//	(* Append sample digital inputs *)
//	FOR iLoop := 0 TO 19 DO
//		fbVisuControl.MR_AppendSafeInput(ifSafeInput := stShell.stPlatform.ref_fbMachineControler.SafeInputs[iLoop]);
//	END_FOR
	
//	(* Append sample digital outputs *)
//	FOR iLoop := 0 TO 19 DO
//		fbVisuControl.MR_AppendSafeOutput(ifSafeOutput := stShell.stPlatform.ref_fbMachineControler.SafeOutputs[iLoop]);
//	END_FOR
	
//	(* Append sample double coil cylinders *)
//	FOR iLoop := 0 TO 9 DO
//		fbVisuControl.MR_AppendCylinder( 	ifCylinder 			:= stShell.stPlatform.ref_fbMachineControler.DoubleCoilCylinders[iLoop],
//											eCylinderType 		:= CYLINDER_TYPE_DOUBLE_COIL,
//											sActiveDescription	:= 'Active',
//											sHomeDescription	:= 'Home');
//	END_FOR
	
//	(* Append sample single coil cylinders *)
//	FOR iLoop := 0 TO 9 DO
//		fbVisuControl.MR_AppendCylinder( 	ifCylinder 			:= stShell.stPlatform.ref_fbMachineControler.SingleCoilCylinders[iLoop],
//											eCylinderType 		:= CYLINDER_TYPE_SINGLE_COIL,
//											sActiveDescription 	:= 'Active',
//											sHomeDescription 	:= 'Home');
//	END_FOR
	(* Append sample scara robot *)
	//FOR iLoop := 0 TO 4 DO
		fbVisuControl.MR_AppendRobot(	ifRobot 	:= stShell.stPlatform.ref_fbMachineControler.Robots,
										eRobotType	:= ROBOT_TYPE_MITSUBISHI_SCARA);
	//END_FOR
	
//	(* Append sample 6 axis robot *)
//	FOR iLoop := 5 TO 9 DO
//		fbVisuControl.MR_AppendRobot(	ifRobot 	:= stShell.stPlatform.ref_fbMachineControler.Robots[iLoop],
//										eRobotType	:= ROBOT_TYPE_MITSUBISHI_6_AXIS);
//	END_FOR
	
//	(* Append sample axes *)
//	FOR iLoop := 0 TO 19 DO
//		fbVisuControl.MR_AppendAxis(	ifMotor		:= stShell.stPlatform.ref_fbMachineControler.Axes[iLoop],
//										eMotorType	:= AXIS_TYPE_BECKHOFF_XTS_MOVER);
//	END_FOR

	(* Set assignamnet done bit *)
	stShell.stFlags.bVisuCtrlAssignamentsDone := TRUE;
END_IF

(* Start running Visu Controler if all other controlers are assigned *)
IF stShell.stFlags.bVisuCtrlAssignamentsDone THEN
	fbVisuControl();
END_IF

END_PROGRAM

// ---- POUs/Machine/Visu Control/FB_VisuControl.TcPOU
FUNCTION_BLOCK FB_VisuControl EXTENDS FB_UniversalVisu
VAR
END_VAR

bBackupRestoreDisabled := TRUE;
SUPER^();

METHOD PROTECTED  MS_Emergency
;
END_METHOD

END_FUNCTION_BLOCK

// ---- POUs/Libs/Platform/Universal Visu/FB_UniversalVisu.TcPOU
(* 
:Description: This function block is base for of machine HMI module in all projects.
*)
FUNCTION_BLOCK ABSTRACT FB_UniversalVisu
VAR
	(* --- Auxilary variables --- *)
	bFirstCycle 						: BOOL := TRUE;	(*  *)
	iLoop								: USINT;		(*  *)
	iLoop2								: USINT;		(*  *)
	                        			
	(* --- Header --- *)    			
	sMachineName						: STRING;	(*  *)
	sSoftwareVersion					: STRING;	(*  *)
	sCurrentDate						: STRING;	(*  *)
	sCurrentTime						: STRING;	(*  *)
	sCurrentUser						: STRING;	(*  *)
	sCurrentRecipe						: STRING;	(*  *)
                            			
	iActiveAlarms						: UDINT;				(*  *)
	iActiveCriticals 					: REFERENCE TO UDINT;	(*  *)
	iActvieErrors						: REFERENCE TO UDINT;	(*  *)
	iActiveWarrnings					: REFERENCE TO UDINT;	(*  *)
	
	(* --- Navigation bar --- *)
	btnInit								: BOOL;		(*  *)
	btnReset							: BOOL;		(*  *)
	btnManual 							: BOOL;		(*  *)
	btnAuto								: BOOL;		(*  *)
	btnAbort 							: BOOL;		(*  *)
	btnStart 							: BOOL;		(*  *)
	btnStop 							: BOOL;		(*  *)
	btnStepMode 						: BOOL;		(*  *)
	btnBack 							: BOOL;		(*  *)
	                    			
	bInit								: BOOL;		(*  *)
	bReset								: BOOL;		(*  *)
	bAbort 								: BOOL;		(*  *)
	
	(* --- Auxilary navigation bar --- *)
	btnCloseHMI							: BOOL;		(*  *)
	btnAlarms							: BOOL;		(*  *)
	btnRecipes							: BOOL;		(*  *)
	btnLogIn							: BOOL;		(*  *)
	btnLogOut							: BOOL;		(*  *)
	btnChangePass						: BOOL;		(*  *)
	btnLights							: BOOL;		(*  *)
	                        			
	sCloseHMIFileName					: STRING := 'C:\Windows\System32\cmd.exe';	(*  *) //'C:\HMI Utility\CloseHMI.bat',
	sCloseHMIParameters					: STRING := 'taskkill /IM Tc3PlcHmi.exe /F';	(*  *) //'C:\HMI Utility',
	
	(* --- Initialization indicators --- *)
	iInitProgressBar 					: USINT;			(*  *)
	
	(* --- Manual mode --- *)	
	btnManualCylinder					: BOOL;				(*  *)
	btnManualAxis						: BOOL;				(*  *)
	btnManualSafety						: BOOL;				(*  *)
	btnManualOthers						: BOOL;				(*  *)
	btnManualOutputs					: BOOL;				(*  *)
	btnManualInputs						: BOOL;				(*  *)
	btnManualRobots						: BOOL;				(*  *)
	                        			
	bManualCylinderDisabled				: BOOL := FALSE;	(*  *)
	bManualAxisDisabled					: BOOL := FALSE;	(*  *)
	bManualInputsDisabled				: BOOL := FALSE;	(*  *)
	bManualOutputsDisabled				: BOOL := FALSE;	(*  *)
	bManualSafetyDisabled				: BOOL := FALSE;	(*  *)
	bManualOthersDisabled				: BOOL := FALSE;	(*  *)
	bManualRobotDisabled				: BOOL := FALSE;	(*  *)	
	
	btnNext								: BOOL;			(* *)
	btnPrevious							: BOOL;			(* *)
	btnNextInput						: BOOL;			(* *)
	btnPreviousInput					: BOOL;			(* *)
	btnNextOutput						: BOOL;			(* *)
	btnPreviousOutput					: BOOL;			(*  *)
                                    	
	bNextInvisible						: BOOL;			(*  *)
	bPreviousInvisible					: BOOL;			(*  *)
	bNextInvisibleInput					: BOOL;			(*  *)
	bPreviousInvisibleInput				: BOOL;			(*  *)
	bNextInvisibleOutput				: BOOL;			(*  *)
	bPreviousInvisibleOutput			: BOOL;			(*  *)
	                                	
	iSelectedCylinderPageIndex			: USINT := 0;	(*  *)
	iSelectedAxisPageIndex				: USINT := 0;	(*  *)
	iSelectedInputPageIndex 			: USINT := 0;	(*  *)
	iSelectedOutputPageIndex			: USINT := 0;	(*  *)
	iSelectedSafeInputPageIndex 		: USINT := 0;	(*  *)
	iSelectedSafeOutputPageIndex		: USINT := 0;	(*  *)
	iSelectedRobotPageIndex				: USINT := 0;	(*  *)
	
	iCylinderIndex						: USINT := 0;	(*  *)
	iAxisIndex							: USINT := 0;	(*  *)
	iInputIndex							: USINT := 0;	(*  *)
	iOutputIndex						: USINT := 0;	(*  *)
	iSafeInputIndex						: USINT := 0;	(*  *)
	iSafeOutputIndex					: USINT := 0;	(*  *)
	iRobotIndex							: USINT := 0;	(*  *)
                            			
	iCylinderPageIndex					: USINT := 0;	(*  *)
	iAxisPageIndex						: USINT := 0;	(*  *)
	iInputPageIndex						: USINT := 0;	(*  *)
	iOutputPageIndex					: USINT := 0;	(*  *)
	iSafeInputPageIndex					: USINT := 0;	(*  *)
	iSafeOutputPageIndex				: USINT := 0;	(*  *)
	iRobotPageIndex						: USINT := 0;	(*  *)
	                        			
	iCylinderFrameIndex					: USINT := 0;	(*  *)
	iAxisFrameIndex						: USINT := 0;	(*  *)
	iInputFrameIndex					: USINT := 0;	(*  *)
	iOutputFrameIndex					: USINT := 0;	(*  *)
	iSafeInputFrameIndex				: USINT := 0;	(*  *)
	iSafeOutputFrameIndex				: USINT := 0;	(*  *)
	iRobotFrameIndex					: USINT := 0;	(*  *)
                            			
	arrCylinderFrameEmpty 				: ARRAY [0..iMAX_CYLINDER_PAGES-1] OF ARRAY [0..iCYLINDERS_PER_PAGE-1] OF BOOL;								(*  *)
	arrAxisFrameEmpty					: ARRAY [0..iMAX_AXIS_PAGES-1] OF ARRAY [0..iAXIS_PER_PAGE-1] OF BOOL;										(*  *)
	arrInputFrameEmpty					: ARRAY [0..iMAX_INPUT_PAGES-1] OF ARRAY [0..iINPUTS_PER_PAGE-1] OF BOOL;									(*  *)
	arrOutputFrameEmpty					: ARRAY [0..iMAX_OUTPUT_PAGES-1] OF ARRAY [0..iOUTPUTS_PER_PAGE-1] OF BOOL;									(*  *)
	arrSafeInputFrameEmpty				: ARRAY [0..iMAX_SAFE_INPUT_PAGES-1] OF ARRAY [0..iSAFE_INPUTS_PER_PAGE-1] OF BOOL;							(*  *)
	arrSafeOutputFrameEmpty				: ARRAY [0..iMAX_SAFE_OUTPUT_PAGES-1] OF ARRAY [0..iSAFE_OUTPUTS_PER_PAGE-1] OF BOOL;						(*  *)
	arrRobotFrameEmpty					: ARRAY [0..iMAX_ROBOT_PAGES-1] OF ARRAY [0..iROBOTS_PER_PAGE-1] OF BOOL;									(*  *)
	                        			
	arrCylinderFrame					: ARRAY [0..iMAX_CYLINDER_PAGES-1] OF ARRAY [0..iCYLINDERS_PER_PAGE-1] OF ST_VisuCtrlCylinderFrame;			(*  *)
	arrAxisFrame						: ARRAY [0..iMAX_AXIS_PAGES-1] OF ARRAY [0..iAXIS_PER_PAGE-1] OF ST_VisuCtrlAxisFrame;						(*  *)
	arrInputFrame						: ARRAY [0..iMAX_INPUT_PAGES-1] OF ARRAY [0..iINPUTS_PER_PAGE-1] OF ST_VisuCtrlInputFrame;					(*  *)
	arrOutputFrame						: ARRAY [0..iMAX_OUTPUT_PAGES-1] OF ARRAY [0..iOUTPUTS_PER_PAGE-1] OF ST_VisuCtrlOutputFrame;				(*  *)
	arrSafeInputFrame					: ARRAY	[0..iMAX_SAFE_INPUT_PAGES-1] OF ARRAY [0..iSAFE_INPUTS_PER_PAGE-1] OF ST_VisuCtrlInputFrame;		(*  *)
	arrSafeOutputFrame					: ARRAY [0..iMAX_SAFE_OUTPUT_PAGES-1] OF ARRAY [0..iSAFE_OUTPUTS_PER_PAGE-1] OF ST_VisuCtrlOutputFrame;		(*  *)
	arrRobotFrame						: ARRAY [0..iMAX_ROBOT_PAGES-1] OF ARRAY [0..iROBOTS_PER_PAGE-1] OF ST_VisuCtrlRobotFrame;					(*  *)
		                    			
	arrCylinderState					: ARRAY [0..iMAX_CYLINDER_PAGES-1] OF ARRAY [0..iCYLINDERS_PER_PAGE-1] OF E_VisuCtrlSingleCylinderState;	(*  *)
	arrAxisState						: ARRAY [0..iMAX_AXIS_PAGES-1] OF ARRAY [0..iAXIS_PER_PAGE-1] OF E_VisuCtrlSingleAxisState;					(*  *)
	arrRobotState						: ARRAY [0..iMAX_ROBOT_PAGES-1] OF ARRAY [0..iROBOTS_PER_PAGE-1] OF E_VisuCtrlSingleRobotState;				(*  *)
                            			
	arrCylinderLink						: ARRAY [0..iMAX_CYLINDER_PAGES-1] OF ARRAY [0..iCYLINDERS_PER_PAGE-1] OF I_UniversalCylinder;				(*  *)
	arrAxisLink							: ARRAY [0..iMAX_AXIS_PAGES-1] OF ARRAY [0..iAXIS_PER_PAGE-1] OF I_UniversalAxis;							(*  *)
	arrInputLink						: ARRAY [0..iMAX_INPUT_PAGES-1] OF ARRAY [0..iINPUTS_PER_PAGE-1] OF I_DigitalInput;							(*  *)
	arrOutputLink						: ARRAY [0..iMAX_OUTPUT_PAGES-1] OF ARRAY [0..iOUTPUTS_PER_PAGE-1] OF I_DigitalOutput;						(*  *)
	arrSafeInputLink					: ARRAY	[0..iMAX_SAFE_INPUT_PAGES-1] OF ARRAY [0..iSAFE_INPUTS_PER_PAGE-1] OF I_DigitalInput;				(*  *)
	arrSafeOutputLink					: ARRAY [0..iMAX_SAFE_OUTPUT_PAGES-1] OF ARRAY [0..iSAFE_OUTPUTS_PER_PAGE-1] OF I_DigitalOutput;			(*  *)
	arrRobotLink						: ARRAY [0..iMAX_ROBOT_PAGES-1] OF ARRAY [0..iROBOTS_PER_PAGE-1] OF I_CR800EtherCAT;						(*  *)
	
	ifUniversalMachineLink				: I_UniversalMachine;	(*  *)
	ifRecipesManager					: I_RecipesManager;		(*  *)
	ifAlarmControler					: I_AlarmControler;		(*  *)
	
	(* --- Alarm page --- *)
	btnClearAll							: BOOL;	(*  *)
	btnExport							: BOOL;	(*  *)
	
	(* --- Recipes page --- *)
	(* Recipe control - buttons *)
	btnCreate							: BOOL;	(* Create recipe button *)
	btnSelect							: BOOL;	(* Select recipe from table button*)
	btnLoad								: BOOL;	(* Load recipe from file button *)
	btnRead								: BOOL;	(* Read recipe to file button *)
	btnReload 							: BOOL;	(* Reload recipes button *)
	btnBackup							: BOOL;	(* Backup recipes to external directory button *)
	btnRestore							: BOOL;	(* Restore recipes from external directory button *)
	btnRemove							: BOOL;	(* Remove recipe from the file *)
	btnReloadExternal					: BOOL;	(* Reload recipes button *)
	btnRecipeNext						: BOOL;	(* Go to next page with recipe parameters *)
	btnRecipePrevious					: BOOL;	(* Go to previous page with recipe parameters *)
	btnHmiClose							: BOOL;
	
	bUpdateVisuElements					: BOOL; (* For function block extending purposes (updating some visualisation elements after loading recipes) *)

	
	(* Recipe control - visibility *)
	bReloadInvisible					: BOOL;	(* Makes reload button invisible *)
	bRecipeNextInvisible				: BOOL;	(* Makes next button invisible *)
	bRecipePreviousInvisible			: BOOL;	(* Makes previous button invisible *)
	bRecipeCreateInvisible				: BOOL;	(* Makes create group box invisible *)
	bRecipeBackupRestoreInvisible		: BOOL;	(* Makes backup and restore group box invisible *)
	bNoRecipeSelected					: BOOL;
	
	(* Recipe control - control disabled *)
	bCreateRecipeDisabled				: BOOL;	(* Disable access to create recipe group box *)
	bBackupRestoreDisabled				: BOOL;	(* Disable access to backup and restore group box *)
	
	(* Recipe control - status *)
	bRecipesManagerError				: REFERENCE TO BOOL;					(* Error occured while executing last command *)
	eRecipesManagerReturns				: REFERENCE TO E_RecipesManagerReturns;	(* Result of last executed command *)
	
	(* Recipe control - parameters for recipes manager *)
	iSelectedRecipe						: INT;												(* Number of selected row in Available Recipes table *)
	sRecipeDefinition					: REFERENCE TO STRING;								(* Name of current recipe definition *)
	sSelectedRecipe						: STRING;											(* Current selected recipe name - changes affter trigger from btnSelect *)
	sNewRecipeName						: STRING;											(* Name for new recipe *)
	sBackupStoragePath					: STRING;											(* Path for backup/restoring of recipes *)
	arrRecipesNames						: REFERENCE TO ARRAY[0..127] OF STRING;				(* Names of all detected recipes *)
	sBackupRestoreRecipeName			: STRING;
		
	(* Recipe control - parameters frame generator *)
	iRecipeParameterIndex 				: USINT := 0;	(*  *)
	iRecipeParameterFrameIndex			: USINT := 0;	(*  *)	
	iRecipeParameterPageIndex			: USINT := 0;	(*  *)
	iSelectedRecipeParameterPageIndex	: USINT := 0;	(*  *)
	
	arrRecipeParameterFrameEmpty 		: ARRAY [0..iMAX_NUMBER_OF_RECIPES-1] OF ARRAY [0..iRECIPE_PARAMETERS_PER_PAGE-1] OF BOOL;							(*  *)
	arrRecipeParameterLink				: ARRAY [0..iMAX_NUMBER_OF_RECIPES-1] OF ARRAY [0..iRECIPE_PARAMETERS_PER_PAGE-1] OF I_RecipeParameter;				(*  *)
	arrRecipeParameterFrameData			: ARRAY [0..iMAX_NUMBER_OF_RECIPES-1] OF ARRAY [0..iRECIPE_PARAMETERS_PER_PAGE-1] OF ST_VisuCtrlRecipeParameter;	(*  *)
	arrRecipeParameterFrameType			: ARRAY [0..iMAX_NUMBER_OF_RECIPES-1] OF ARRAY [0..iRECIPE_PARAMETERS_PER_PAGE-1] OF E_VisuCtrlRecipeParameterType;	(*  *)
	
	(* --- Shell state machines --- *)
	eUniversalMachineCtrlState			: E_VisuCtrUniversalMachineState;		(*  *)
	eRecipesManagerState				: E_VisuCtrlRecipesManagerState;			(* Current state of Recipe Manager *)
	eAlarmCtrlState						: E_VisuCtrlAlarmControlState;			(* Current state of Alarm Controler *)
	
	(* --- Screen selectors --- *)
	eCurrentScreen						: E_VisuCtrlPageState;					(* Main page selector *)
	eLastScreen							: E_VisuCtrlPageState;					(* Last screen before change to auxilary screen *)
	eCurrentNavigation					: E_VisuCtrlNavBarState;				(* Navigation bar selector *)
	
	(* --- HMI buttons flags --- *)
	bStartDisable 						: BOOL;
	bStopDisable						: BOOL	:= TRUE;
	bVisNotInit 						: BOOL	:= TRUE;	
	bVisLogIn							: BOOL;
	bVisLogOut 							: BOOL	:= TRUE;	
	bVisHmiClose						: BOOL;
	bRecipeButtonDisabled				: BOOL;
	bModeSwitchButtonDisabled			: BOOL;
	                        			
	fbHmiClose							: NT_StartProcess;
END_VAR
(*
Version history:

+-------------+------------+----------------+----------+------------------------------------------+
|Date         | Version    | created under  | Author   | Remark                                   |
+=============+============+================+==========+==========================================+
|2022-03      | 1.0.0.0    | V3.1.4024.22   | ADBO     | Function block created                   |
+-------------+------------+----------------+----------+------------------------------------------+

*)

IF bFirstCycle THEN
	bFirstCycle := FALSE;
	(* Assign alarm references *)
	iActiveCriticals	REF= ifAlarmControler.ActiveCritical;
	iActvieErrors 		REF= ifAlarmControler.ActiveError;
	iActiveWarrnings	REF= ifAlarmControler.ActiveWarrning;
	
	(* Assign recipes references *)
	bRecipesManagerError 	REF= ifRecipesManager.Error;
	arrRecipesNames 		REF= ifRecipesManager.RecipesNames;
	eRecipesManagerReturns 	REF= ifRecipesManager.LastResult;
	sRecipeDefinition 		REF= ifRecipesManager.RecipesDefinition;
	
	(* --- Mark unused frames - saves CPU resources --- *)
	(* Cylinder frames *)
	FOR iLoop := 0 TO iMAX_CYLINDER_PAGES-1 DO
		FOR iLoop2 := 0 TO iCYLINDERS_PER_PAGE-1 DO
			IF arrCylinderLink[iLoop][iLoop2] = 0 THEN
				arrCylinderFrameEmpty[iLoop][iLoop2] := TRUE;
			END_IF
		END_FOR
	END_FOR
	
	(* Motor frames *)
	FOR iLoop := 0 TO iMAX_AXIS_PAGES-1 DO
		FOR iLoop2 := 0 TO iAXIS_PER_PAGE-1 DO
			IF arrAxisLink[iLoop][iLoop2] = 0 THEN
				arrAxisFrameEmpty[iLoop][iLoop2] := TRUE;
			END_IF
		END_FOR
	END_FOR
	
	(* Input frames *)
	FOR iLoop := 0 TO iMAX_INPUT_PAGES-1 DO
		FOR iLoop2 := 0 TO iINPUTS_PER_PAGE-1 DO
			IF arrInputLink[iLoop][iLoop2] = 0 THEN
				arrInputFrameEmpty[iLoop][iLoop2] := TRUE;
			END_IF
		END_FOR
	END_FOR
	
	(* Output frames *)
	FOR iLoop := 0 TO iMAX_OUTPUT_PAGES-1 DO
		FOR iLoop2 := 0 TO iOUTPUTS_PER_PAGE-1 DO
			IF arrOutputLink[iLoop][iLoop2] = 0 THEN
				arrOutputFrameEmpty[iLoop][iLoop2] := TRUE;
			END_IF
		END_FOR
	END_FOR
	
	(* Safe input frames *)
	FOR iLoop := 0 TO iMAX_SAFE_INPUT_PAGES-1 DO
		FOR iLoop2 := 0 TO iSAFE_INPUTS_PER_PAGE-1 DO
			IF arrSafeInputLink[iLoop][iLoop2] = 0 THEN
				arrSafeInputFrameEmpty[iLoop][iLoop2] := TRUE;
			END_IF
		END_FOR
	END_FOR
	
	(* Safe output frames *)
	FOR iLoop := 0 TO iMAX_SAFE_OUtPUT_PAGES-1 DO
		FOR iLoop2 := 0 TO iSAFE_OUtPUTS_PER_PAGE-1 DO
			IF arrSafeOutputLink[iLoop][iLoop2] = 0 THEN
				arrSafeOutputFrameEmpty[iLoop][iLoop2] := TRUE;
			END_IF
		END_FOR
	END_FOR
	
	(* Robot frames *)
	FOR iLoop := 0 TO iMAX_ROBOT_PAGES-1 DO
		FOR iLoop2 := 0 TO iROBOTS_PER_PAGE-1 DO
			IF arrRobotLink[iLoop][iLoop2] = 0 THEN
				arrRobotFrameEmpty[iLoop][iLoop2] := TRUE;
			END_IF
		END_FOR
	END_FOR
	
	(* Universal fixture frames *)
	//To-do
	
	(* Tcp-Server frames *)
	// To do
	
	(* Tcp-Client frames*)
	// To do
	
	(* Robot frames *)
	FOR iLoop := 0 TO iMAX_ROBOT_PAGES - 1 DO
		FOR iLoop2 := 0 TO iROBOTS_PER_PAGE - 1 DO
			IF arrRobotLink[iLoop][iLoop2] = 0 THEN
				arrRobotFrameEmpty[iLoop][iLoop2] := TRUE;
			END_IF
		END_FOR
	END_FOR
	
	(* Recipe parameters frames *)
	FOR iLoop := 0 TO iMAX_RECIPES_PAGES-1 DO
		FOR iLoop2 := 0 TO iRECIPE_PARAMETERS_PER_PAGE-1 DO
			IF arrRecipeParameterLink[iLoop][iLoop2] = 0 THEN
				arrRecipeParameterFrameEmpty[iLoop][iLoop2] := TRUE;
			END_IF
		END_FOR
	END_FOR
	
END_IF

(* Get current logged in user *)
IF btnLogIn AND LEN(WSTRING_TO_STRING(VisuUserManagement.VisuElems.CurrentFullUserName)) <> 0 THEN
	sCurrentUser := WSTRING_TO_STRING(VisuUserManagement.VisuElems.CurrentFullUserName);
	btnLogIn := FALSE;
ELSIF btnLogOut THEN
	MEMSET(ADR(sCurrentUser),0,SIZEOF(sCurrentUser));
	btnLogOut := FALSE;
END_IF

(* LogIn and LogOut button status flags *)
IF LEN(sCurrentUser) <> 0 THEN 
	bVisLogIn := TRUE;
	bVisLogOut:= FALSE;
	
ELSE
	bVisLogIn := FALSE;
	bVisLogOut:= TRUE;
	
END_IF

fbHmiClose(
	NETID			:= '',
	PATHSTR			:= 'C:\WINDOWS\system32\taskkill.exe' ,
	DIRNAME			:= '' ,
	COMNDLINE		:= '/t /f /IM Tc3PlcHmi.exe' , 
	START			:= btnHmiClose,
	ERRID			=> );

IF fbHmiClose.BUSY THEN		
	btnHmiClose := FALSE;	
END_IF

(* Get time and date *)
sCurrentDate := FUN_TimestructToDate(fbMachineTime.systemTime);
sCurrentTime := FUN_TimestructToTime(fbMachineTime.systemTime);
sCurrentTime := LEFT(STR := sCurrentTime, SIZE := (LEN(sCurrentTime)-4));

(* Universal switch to Alarms and Recipes page *)
IF btnRecipes THEN
	btnRecipes := FALSE;
	IF eCurrentScreen <> SCREEN_RECIPES AND eCurrentScreen <> SCREEN_ALARMS THEN
		eLastScreen := eCurrentScreen;
	END_IF
	eCurrentScreen := SCREEN_RECIPES;
	
ELSIF btnAlarms THEN
	btnAlarms := FALSE;
	IF eCurrentScreen <> SCREEN_RECIPES AND eCurrentScreen <> SCREEN_ALARMS THEN
		eLastScreen := eCurrentScreen;
	END_IF
	eCurrentScreen := SCREEN_ALARMS;
END_IF

(* Universal change to Abort - Reset mode *)
IF btnAbort THEN
	btnAbort := FALSE;
	eUniversalMachineCtrlState := VISU_CTRL_UNIVERSAL_MACHINE_ABORT;
	eAlarmCtrlState := VISU_CTRL_ALARM_CONTROLER_ABORT;
	eRecipesManagerState := VISU_CTRL_RECIPE_MANAGER_ABORT;
	eRecipesManagerState := VISU_CTRL_RECIPE_MANAGER_INIT;
	eCurrentScreen := SCREEN_ABORTING;
			
ELSIF btnReset THEN
	btnReset := FALSE;
	eUniversalMachineCtrlState := VISU_CTRL_UNIVERSAL_MACHINE_RESET;
END_IF

(* --- Alarm system control via shared interface --- *)
M_AlarmControler();

(* --- Recipes manager control via shared interface --- *)
M_RecipeManager();

(* --- Universal Machine control via shared interface ---*)
M_MachineControler();

(* --- Generic content control state machine --- *)
StateMachine();

PROPERTY Abort : REFERENCE TO BOOL
GET
Abort REF= btnAbort;
END_GET
END_PROPERTY

PROPERTY AutoMode : REFERENCE TO BOOL
GET
AutoMode REF= btnAuto;
END_GET
END_PROPERTY

PROPERTY Back : REFERENCE TO BOOL
GET
Back REF= btnBack;
END_GET
END_PROPERTY

PROPERTY Init : REFERENCE TO BOOL
GET
Init REF= btnInit;
END_GET
END_PROPERTY

METHOD PROTECTED M_AlarmControler
(* --- Active alarms counter --- *)
(*iActiveCriticals := ifAlarmControler.ActiveCritical;
iActvieErrors := ifAlarmControler.ActiveError;
iActiveWarrnings := ifAlarmControler.ActiveWarrning;*)
iActiveAlarms := iActvieErrors + iActiveCriticals;

(* Main alarm control via HMI *)
CASE eAlarmCtrlState OF
	VISU_CTRL_ALARM_CONTROLER_WAIT_FOR_CMD:
		IF btnInit THEN
			eAlarmCtrlState := VISU_CTRL_ALARM_CONTROLER_INIT;
			
		ELSIF btnClearAll THEN
			eAlarmCtrlState := VISU_CTRL_ALARM_CONTROLER_CLEAR_ALL; 
			
		ELSIF btnExport THEN
			eAlarmCtrlState := VISU_CTRL_ALARM_CONTTOLER_EXPORT;
			
		END_IF
		
	VISU_CTRL_ALARM_CONTROLER_INIT:
		ifAlarmControler.MR_Init();
		
		IF ifAlarmControler.Active THEN
			eAlarmCtrlState := VISU_CTRL_ALARM_CONTROLER_WAIT_FOR_CMD;
		END_IF
		
	VISU_CTRL_ALARM_CONTROLER_CLEAR_ALL:
		ifAlarmControler.MR_ClearAll(bResetConfirmation := TRUE);
		
		IF NOT ifAlarmControler.Busy THEN
			eAlarmCtrlState := VISU_CTRL_ALARM_CONTROLER_WAIT_FOR_CMD;
		END_IF
	
	VISU_CTRL_ALARM_CONTTOLER_EXPORT:
		ifAlarmControler.MR_Export();
		
		IF NOT ifAlarmControler.Busy THEN
			eAlarmCtrlState := VISU_CTRL_ALARM_CONTROLER_WAIT_FOR_CMD;
		END_IF
		
	VISU_CTRL_ALARM_CONTROLER_ABORT:
		ifAlarmControler.MR_Abort();
		
		IF NOT ifAlarmControler.Active THEN
			eAlarmCtrlState := VISU_CTRL_ALARM_CONTROLER_WAIT_FOR_CMD;
		END_IF
		
END_CASE
END_METHOD

METHOD M_MachineControler : BOOL
(* Main machine control via HMI *)
IF NOT ifUniversalMachineLink.Running THEN
	bStartDisable := FALSE;
	bStopDisable := TRUE;
ELSE
	bStartDisable := TRUE;
	bStopDisable := FALSE;
END_IF

CASE eUniversalMachineCtrlState OF
	VISU_CTRL_UNIVERSAL_MACHINE_WAIT_FOR_CMD:
		IF btnInit THEN
			eUniversalMachineCtrlState := VISU_CTRL_UNIVERSAL_MACHINE_INIT;
			
		ELSIF btnStart THEN
			eUniversalMachineCtrlState := VISU_CTRL_UNIVERSAL_MACHINE_START_AUTO;
			
		ELSIF btnStop THEN
			eUniversalMachineCtrlState := VISU_CTRL_UNIVERSAL_MACHINE_STOP_AUTO;
			
		ELSIF btnManual THEN
			eUniversalMachineCtrlState := VISU_CTRL_UNIVERSAL_MACHINE_SWITCH_TO_MANUAL;
			
		ELSIF btnAuto THEN
			eUniversalMachineCtrlState := VISU_CTRL_UNIVERSAL_MACHINE_SWITCH_TO_AUTO;
			
		ELSIF btnAbort THEN
			eUniversalMachineCtrlState := VISU_CTRL_UNIVERSAL_MACHINE_ABORT;
			
		ELSIF btnReset THEN
			eUniversalMachineCtrlState := VISU_CTRL_UNIVERSAL_MACHINE_RESET;			
		END_IF
	
	VISU_CTRL_UNIVERSAL_MACHINE_INIT:
		ifUniversalMachineLink.MR_Init();
		
		IF ifUniversalMachineLink.Active THEN
			bVisNotInit := FALSE;
			bVisHmiClose:= TRUE;
						
			eUniversalMachineCtrlState := VISU_CTRL_UNIVERSAL_MACHINE_WAIT_FOR_CMD;
		END_IF
	
	VISU_CTRL_UNIVERSAL_MACHINE_RESET:
		ifUniversalMachineLink.MR_Reset();
		
		IF NOT ifUniversalMachineLink.Error THEN
			eUniversalMachineCtrlState := VISU_CTRL_UNIVERSAL_MACHINE_WAIT_FOR_CMD;
		END_IF
	
	VISU_CTRL_UNIVERSAL_MACHINE_START_AUTO:
		ifUniversalMachineLink.MR_Start();
		
		IF ifUniversalMachineLink.Running THEN
			eUniversalMachineCtrlState := VISU_CTRL_UNIVERSAL_MACHINE_WAIT_FOR_CMD;
		END_IF
	
	VISU_CTRL_UNIVERSAL_MACHINE_STOP_AUTO:
		ifUniversalMachineLink.MR_Stop();
		
		IF NOT ifUniversalMachineLink.Running THEN
			eUniversalMachineCtrlState := VISU_CTRL_UNIVERSAL_MACHINE_WAIT_FOR_CMD;
		END_IF
		
	VISU_CTRL_UNIVERSAL_MACHINE_SWITCH_TO_MANUAL:
		ifUniversalMachineLink.MR_SwitchToManual();
		
		IF ifUniversalMachineLink.State = MACHINE_STATE_MANUAL THEN
			eUniversalMachineCtrlState := VISU_CTRL_UNIVERSAL_MACHINE_WAIT_FOR_CMD;
		END_IF
	
	VISU_CTRL_UNIVERSAL_MACHINE_SWITCH_TO_AUTO:
		ifUniversalMachineLink.MR_SwitchToAuto();
		
		IF ifUniversalMachineLink.State = MACHINE_STATE_AUTO THEN
			eUniversalMachineCtrlState := VISU_CTRL_UNIVERSAL_MACHINE_WAIT_FOR_CMD;
		END_IF
	
	VISU_CTRL_UNIVERSAL_MACHINE_ABORT:
		ifUniversalMachineLink.MR_Abort();
		
		IF NOT ifUniversalMachineLink.Active THEN
			bVisNotInit := TRUE;
			bVisHmiClose:= FALSE;
			
			eUniversalMachineCtrlState := VISU_CTRL_UNIVERSAL_MACHINE_WAIT_FOR_CMD;
		END_IF
		
END_CASE
END_METHOD

METHOD PROTECTED M_RecipeManager
bRecipesManagerError 	:= ifRecipesManager.Error;
arrRecipesNames 		:= ifRecipesManager.RecipesNames;
eRecipesManagerReturns 	:= ifRecipesManager.LastResult;
sRecipeDefinition 		:= ifRecipesManager.RecipesDefinition;

IF bStartDisable OR bVisNotInit THEN
	bRecipeButtonDisabled := TRUE;
ELSE
	bRecipeButtonDisabled := FALSE;
END_IF

(* Previous page button visiblity control *)
IF iSelectedRecipeParameterPageIndex = 0 THEN
	bRecipePreviousInvisible := TRUE;
ELSE
	bRecipePreviousInvisible := FALSE;
END_IF

IF sSelectedRecipe = '' THEN
	bNoRecipeSelected := TRUE;

ELSE 
	bNoRecipeSelected := FALSE;

END_IF

(* Next page button visibility control *)
IF btnRecipeNext THEN
	btnRecipeNext := FALSE;
	iSelectedRecipeParameterPageIndex := iSelectedRecipeParameterPageIndex + 1;
	
ELSIF btnRecipePrevious THEN
	btnRecipePrevious := FALSE;
	iSelectedRecipeParameterPageIndex := iSelectedRecipeParameterPageIndex - 1;
END_IF

(* Selecting new recipe from table *)
IF btnSelect THEN
	btnSelect := FALSE;
	sSelectedRecipe	:= arrRecipesNames[iSelectedRecipe];
	eRecipesManagerState := VISU_CTRL_RECIPE_MANAGER_RELOAD;
END_IF

(* Main recipe manager control via HMI *)
CASE eRecipesManagerState OF
	VISU_CTRL_RECIPE_MANAGER_WAIT_FOR_CMD:
		IF btnInit THEN
			eRecipesManagerState := VISU_CTRL_RECIPE_MANAGER_INIT;
			
		ELSIF btnCreate THEN
			btnCreate := FALSE;
			eRecipesManagerState := VISU_CTRL_RECIPE_MANAGER_CREATE;
			
		ELSIF btnLoad THEN
			btnLoad := FALSE;
			eRecipesManagerState := VISU_CTRL_RECIPE_MANAGER_LOAD;
			
		ELSIF btnRead THEN
			btnRead := FALSE;
			eRecipesManagerState := VISU_CTRL_RECIPE_MANAGER_READ;
			
		ELSIF btnReload THEN
			btnReload := FALSE;
			eRecipesManagerState := VISU_CTRL_RECIPE_MANAGER_RELOAD;	
						
		ELSIF btnReloadExternal THEN
			btnReloadExternal := FALSE;
			eRecipesManagerState := VISU_CTRL_RECIPE_MANAGER_RELOAD_EXT;
			
		ELSIF btnBackup THEN
			btnBackup := FALSE;
			eRecipesManagerState := VISU_CTRL_RECIPE_MANAGER_BACKUP;
			
		ELSIF btnRestore THEN
			btnRestore := FALSE;
			eRecipesManagerState := VISU_CTRL_RECIPE_MANAGER_RESTORE;
			
		ELSIF btnRemove THEN
			btnRemove := FALSE;
			eRecipesManagerState := VISU_CTRL_RECIPE_MANAGER_REMOVE;
						
		END_IF
		
	VISU_CTRL_RECIPE_MANAGER_INIT:
		ifRecipesManager.MR_Init();
		
		IF ifRecipesManager.Active THEN
			eRecipesManagerState := VISU_CTRL_RECIPE_MANAGER_WAIT_FOR_CMD;
		END_IF
	
	VISU_CTRL_RECIPE_MANAGER_CREATE:
		ifRecipesManager.MR_Create( sRecipesDefinition	:= sRecipeDefinition,
									sRecipeName			:= sNewRecipeName);
									
		IF NOT ifRecipesManager.Busy THEN
			eRecipesManagerState := VISU_CTRL_RECIPE_MANAGER_WAIT_FOR_CMD;
		END_IF
	
	VISU_CTRL_RECIPE_MANAGER_LOAD:
		ifRecipesManager.MR_LoadAndWritte( 	sRecipesDefinition	:= sRecipeDefinition,
											sRecipeName			:= sSelectedRecipe);
									
		IF NOT ifRecipesManager.Busy THEN
			IF NOT ifRecipesManager.Error THEN
				sCurrentRecipe := sSelectedRecipe; 
			END_IF
			
			bUpdateVisuElements := TRUE;
			eRecipesManagerState := VISU_CTRL_RECIPE_MANAGER_WAIT_FOR_CMD;
		END_IF
	
	VISU_CTRL_RECIPE_MANAGER_READ:
		ifRecipesManager.MR_ReadAndSave(	sRecipesDefinition	:= sRecipeDefinition,
											sRecipeName			:= sSelectedRecipe);
									
		IF NOT ifRecipesManager.Busy THEN
			eRecipesManagerState := VISU_CTRL_RECIPE_MANAGER_WAIT_FOR_CMD;
		END_IF
	
	VISU_CTRL_RECIPE_MANAGER_RELOAD:
		ifRecipesManager.MR_Reload( sRecipesDefinition := sRecipeDefinition,
									sRecipeName := sSelectedRecipe);
									
		IF NOT ifRecipesManager.Busy THEN
			eRecipesManagerState := VISU_CTRL_RECIPE_MANAGER_WAIT_FOR_CMD;
		END_IF
		
	VISU_CTRL_RECIPE_MANAGER_RELOAD_EXT:
		ifRecipesManager.MR_ReloadExternal( sRecipesDefinition := sRecipeDefinition,
											sRecipeName := sBackupRestoreRecipeName,
											sBackupStoragePath := sBackupStoragePath);
									
		IF NOT ifRecipesManager.Busy THEN
			eRecipesManagerState := VISU_CTRL_RECIPE_MANAGER_WAIT_FOR_CMD;
		END_IF	
	
	VISU_CTRL_RECIPE_MANAGER_BACKUP:
		ifRecipesManager.MR_Backup(sRecipesDefinition := sRecipeDefinition,
									sRecipeName := sBackupRestoreRecipeName,
									sBackupStoragePath := sBackupStoragePath);
									
		IF NOT ifRecipesManager.Busy THEN
			eRecipesManagerState := VISU_CTRL_RECIPE_MANAGER_WAIT_FOR_CMD;
		END_IF
		
	VISU_CTRL_RECIPE_MANAGER_RESTORE:
		ifRecipesManager.MR_Restore(sRecipesDefinition := sRecipeDefinition,
									sRecipeName := sBackupRestoreRecipeName,
									sBackupStoragePath := sBackupStoragePath);
									
		IF NOT ifRecipesManager.Busy THEN
			IF NOT ifRecipesManager.Error THEN
				sCurrentRecipe := sSelectedRecipe; 
			END_IF
			
			bUpdateVisuElements := TRUE;
			eRecipesManagerState := VISU_CTRL_RECIPE_MANAGER_WAIT_FOR_CMD;
		END_IF
		
	VISU_CTRL_RECIPE_MANAGER_REMOVE:
		ifRecipesManager.MR_Remove( sRecipesDefinition := sRecipeDefinition,
									sRecipeName := sSelectedRecipe);
		
		IF NOT ifRecipesManager.Busy THEN
			eRecipesManagerState := VISU_CTRL_RECIPE_MANAGER_WAIT_FOR_CMD;
		END_IF
	
	VISU_CTRL_RECIPE_MANAGER_ABORT:
		ifRecipesManager.MR_Abort();
		
		IF NOT ifRecipesManager.Active THEN
			eRecipesManagerState := VISU_CTRL_RECIPE_MANAGER_WAIT_FOR_CMD;
		END_IF
	
END_CASE
END_METHOD

PROPERTY ManualMode : REFERENCE TO BOOL
GET
ManualMode REF= btnManual;
END_GET
END_PROPERTY

METHOD MR_AppendAlarmControler : BOOL
VAR_INPUT
	ifAlarmControler : I_AlarmControler;
END_VAR
THIS^.ifAlarmControler := ifAlarmControler;
MR_AppendAlarmControler := TRUE;
END_METHOD

METHOD MR_AppendAxis : BOOL
VAR_INPUT
	ifMotor 	: I_UniversalAxis;
	eMotorType	: E_VisuCtrlAxisImgType;
END_VAR
IF iAxisIndex < iMAX_AXIS_FRAMES THEN
	arrAxisLink[iAxisPageIndex][iAxisFrameIndex] := ifMotor;
	arrAxisFrameEmpty[iAxisPageIndex][iAxisFrameIndex] := FALSE;
	arrAxisFrame[iAxisPageIndex][iAxisFrameIndex].sAxisImage := TO_STRING(eMotorType);
	
	IF iAxisFrameIndex = iAXIS_PER_PAGE - 1 THEN
		iAxisPageIndex := iAxisPageIndex + 1;
		iAxisFrameIndex := 0;
	ELSE
		iAxisFrameIndex := iAxisFrameIndex + 1;
	END_IF	

	iAxisIndex := iAxisIndex + 1;
	MR_AppendAxis := TRUE;
ELSE
	MR_AppendAxis := FALSE;
END_IF
END_METHOD

METHOD MR_AppendCylinder : BOOL
VAR_INPUT
	ifCylinder			: I_UniversalCylinder;
	eCylinderType		: E_VisuCtrlCylinderImgType;
	sActiveDescription	: STRING;
	sHomeDescription	: STRING;
END_VAR
IF iCylinderIndex < iMAX_CYLINDER_FRAMES THEN
	arrCylinderLink[iCylinderPageIndex][iCylinderFrameIndex] := ifCylinder;
	arrCylinderFrameEmpty[iCylinderPageIndex][iCylinderFrameIndex] := FALSE;
	
	arrCylinderFrame[iCylinderPageIndex][iCylinderFrameIndex].sCylinderImage := TO_STRING(eCylinderType);
	arrCylinderFrame[iCylinderPageIndex][iCylinderFrameIndex].sActiveDescription := sActiveDescription;
	arrCylinderFrame[iCylinderPageIndex][iCylinderFrameIndex].sHomeDescription := sHomeDescription;
	
	IF iCylinderFrameIndex = iCYLINDERS_PER_PAGE - 1 THEN
		iCylinderPageIndex := iCylinderPageIndex + 1;
		iCylinderFrameIndex := 0;
	ELSE
		iCylinderFrameIndex := iCylinderFrameIndex + 1;
	END_IF	

	iCylinderIndex := iCylinderIndex + 1;
	MR_AppendCylinder := TRUE;
ELSE
	MR_AppendCylinder := FALSE;
END_IF
END_METHOD

METHOD MR_AppendInput : BOOL
VAR_INPUT
	ifDigitalInput : I_DigitalInput;
END_VAR
IF iInputIndex < iMAX_INPUT_FRAMES THEN
	arrInputLink[iInputPageIndex][iInputFrameIndex] := ifDigitalInput;
	arrInputFrameEmpty[iInputPageIndex][iInputFrameIndex] := FALSE;
	
	IF iInputFrameIndex = iINPUTS_PER_PAGE - 1 THEN
		iInputPageIndex := iInputPageIndex + 1;
		iInputFrameIndex := 0;
	ELSE
		iInputFrameIndex := iInputFrameIndex + 1;
	END_IF	
	
	iInputIndex := iInputIndex + 1;
	MR_AppendInput := TRUE;
ELSE
	MR_AppendInput := FALSE;
END_IF
END_METHOD

METHOD MR_AppendOutput : BOOL
VAR_INPUT
	ifDigitalOutput : I_DigitalOutput;
END_VAR
IF iOutputIndex < iMAX_OUTPUT_FRAMES THEN
	arrOutputLink[iOutputPageIndex][iOutputFrameIndex] := ifDigitalOutput;
	arrOutputFrameEmpty[iOutputPageIndex][iOutputFrameIndex] := FALSE;
	
	IF iOutputFrameIndex = iOUTPUTS_PER_PAGE - 1 THEN
		iOutputPageIndex := iOutputPageIndex + 1;
		iOutputFrameIndex := 0;
	ELSE
		iOutputFrameIndex := iOutputFrameIndex + 1;
	END_IF	

	iOutputIndex := iOutputIndex + 1;
	MR_AppendOutput := TRUE;
ELSE
	MR_AppendOutput := FALSE;
END_IF
END_METHOD

METHOD MR_AppendRecipeParameter : BOOL
VAR_INPUT
	ifRecipeParameter : I_RecipeParameter;
END_VAR
IF iRecipeParameterIndex < iMAX_NUMBER_OF_RECIPES THEN
	arrRecipeParameterLink[iRecipeParameterPageIndex][iRecipeParameterFrameIndex] 		:= ifRecipeParameter;
	arrRecipeParameterFrameEmpty[iRecipeParameterPageIndex][iRecipeParameterFrameIndex] := FALSE;
	arrRecipeParameterFrameType[iRecipeParameterPageIndex][iRecipeParameterFrameIndex]	:= ifRecipeParameter.DataType;
	
	arrRecipeParameterFrameData[iRecipeParameterPageIndex][iRecipeParameterFrameIndex].bValue 		REF= arrRecipeParameterLink[iRecipeParameterPageIndex][iRecipeParameterFrameIndex].BitValue;
	arrRecipeParameterFrameData[iRecipeParameterPageIndex][iRecipeParameterFrameIndex].iValue 		REF= arrRecipeParameterLink[iRecipeParameterPageIndex][iRecipeParameterFrameIndex].IntValue;
	arrRecipeParameterFrameData[iRecipeParameterPageIndex][iRecipeParameterFrameIndex].rValue 		REF= arrRecipeParameterLink[iRecipeParameterPageIndex][iRecipeParameterFrameIndex].RealValue;
	arrRecipeParameterFrameData[iRecipeParameterPageIndex][iRecipeParameterFrameIndex].sValue 		REF= arrRecipeParameterLink[iRecipeParameterPageIndex][iRecipeParameterFrameIndex].StringValue;
	arrRecipeParameterFrameData[iRecipeParameterPageIndex][iRecipeParameterFrameIndex].sName 		REF= arrRecipeParameterLink[iRecipeParameterPageIndex][iRecipeParameterFrameIndex].Name;
	arrRecipeParameterFrameData[iRecipeParameterPageIndex][iRecipeParameterFrameIndex].sFileValue 	REF= arrRecipeParameterLink[iRecipeParameterPageIndex][iRecipeParameterFrameIndex].FileValue;
	
	IF iRecipeParameterFrameIndex = iRECIPE_PARAMETERS_PER_PAGE - 1 THEN
		iRecipeParameterPageIndex := iRecipeParameterPageIndex + 1;
		iRecipeParameterFrameIndex := 0;
	ELSE
		iRecipeParameterFrameIndex := iRecipeParameterFrameIndex + 1;
	END_IF	
	
	iRecipeParameterIndex := iRecipeParameterIndex + 1;
	MR_AppendRecipeParameter := FALSE;
ELSE
	MR_AppendRecipeParameter := FALSE;
END_IF
END_METHOD

METHOD MR_AppendRecipesManager : BOOL
VAR_INPUT
	ifRecipesManager : I_RecipesManager;
END_VAR
THIS^.ifRecipesManager := ifRecipesManager;
MR_AppendRecipesManager := TRUE;
END_METHOD

METHOD MR_AppendRobot : BOOL
VAR_INPUT
	ifRobot				: I_CR800EtherCAT;
	eRobotType			: E_VisuCtrlRobotImgType;
//	sErrorDescription	: STRING;
END_VAR
IF iRobotIndex < iMAX_ROBOT_FRAMES THEN
	arrRobotLink[iRobotPageIndex][iRobotFrameIndex] := ifRobot;
	arrRobotFrameEmpty[iRobotPageIndex][iRobotFrameIndex] := FALSE;
	arrRobotFrame[iRobotPageIndex][iRobotFrameIndex].sRobotImage := TO_STRING(eRobotType);
	
	IF iRobotFrameIndex = iROBOTS_PER_PAGE - 1 THEN
		iRobotPageIndex := iRobotPageIndex + 1;
		iRobotFrameIndex := 0;
	ELSE
		iRobotFrameIndex := iRobotFrameIndex + 1;
	END_IF	

	iRobotIndex := iRobotIndex + 1;
	MR_AppendRobot := TRUE;
ELSE
	MR_AppendRobot := FALSE;
END_IF
END_METHOD

METHOD MR_AppendSafeInput : BOOL
VAR_INPUT
	ifSafeInput : I_DigitalInput;
END_VAR
IF iSafeInputIndex < iMAX_SAFE_INPUT_FRAMES THEN
	arrSafeInputLink[iSafeInputPageIndex][iSafeInputFrameIndex] := ifSafeInput;
	arrSafeInputFrameEmpty[iSafeInputPageIndex][iSafeInputFrameIndex] := FALSE;
	
	IF iSafeInputFrameIndex = iSAFE_INPUTS_PER_PAGE - 1 THEN
		iSafeInputPageIndex := iSafeInputPageIndex + 1;
		iSafeInputFrameIndex := 0;
	ELSE
		iSafeInputFrameIndex := iSafeInputFrameIndex + 1;
	END_IF	
	
	iSafeInputIndex := iSafeInputIndex + 1;
	MR_AppendSafeInput := TRUE;
ELSE
	MR_AppendSafeInput := FALSE;
END_IF
END_METHOD

METHOD MR_AppendSafeOutput : BOOL
VAR_INPUT
	ifSafeOutput : I_DigitalOutput;
END_VAR
IF iSafeOutputIndex < iMAX_SAFE_OUTPUT_FRAMES THEN
	arrSafeOutputLink[iSafeOutputPageIndex][iSafeOutputFrameIndex] := ifSafeOutput;
	arrSafeOutputFrameEmpty[iSafeOutputPageIndex][iSafeOutputFrameIndex] := FALSE;
	
	IF iSafeOutputFrameIndex = iSAFE_OUTPUTS_PER_PAGE - 1 THEN
		iSafeOutputPageIndex := iSafeOutputPageIndex + 1;
		iSafeOutputFrameIndex := 0;
	ELSE
		iSafeOutputFrameIndex := iSafeOutputFrameIndex + 1;
	END_IF		

	iSafeOutputIndex := iSafeOutputIndex + 1;
	MR_AppendSafeOutput := TRUE;
ELSE
	MR_AppendSafeOutput := FALSE;
END_IF
END_METHOD

METHOD MR_AppendUniversalMachine : BOOL
VAR_INPUT
	ifMachine : I_UniversalMachine;
END_VAR
THIS^.ifUniversalMachineLink := ifMachine;
MR_AppendUniversalMachine := TRUE;
END_METHOD

METHOD MR_FirstCycle : BOOL
VAR_INPUT
	sMachineName : STRING;
	sSoftwareVersion : STRING;
END_VAR
THIS^.sMachineName := sMachineName;
THIS^.sSoftwareVersion := sSoftwareVersion;
END_METHOD

METHOD PROTECTED MS_Aborting
VAR_INPUT
END_VAR
eCurrentNavigation := NAVIGATION_EMPTY;

IF ifUniversalMachineLink.State = MACHINE_STATE_UNINITIALIZED THEN
	eCurrentScreen := SCREEN_UNINITIALIZED;
	
ELSIF ifUniversalMachineLink.State = MACHINE_STATE_EMERGENCY THEN
	eCurrentScreen := SCREEN_EMERGENCY;
	
END_IF
END_METHOD

METHOD PROTECTED MS_Alarms
VAR_INPUT
END_VAR
eCurrentNavigation := NAVIGATION_UTILITIES;

IF btnBack THEN
	btnBack := FALSE;
	eCurrentScreen := eLastScreen;
END_IF
END_METHOD

METHOD PROTECTED MS_Auto
VAR_INPUT
END_VAR
eCurrentNavigation := NAVIGATION_AUTO;

IF ifUniversalMachineLink.State = MACHINE_STATE_ABORTING THEN
	eCurrentScreen := SCREEN_ABORTING;	

ELSIF ifUniversalMachineLink.State = MACHINE_STATE_AUTO_TO_MANUAL THEN
	eCurrentScreen := SCREEN_MODE_CHANGE;
	
	IF iOutputIndex > 0 THEN
		FOR iLoop := 0 TO iOUTPUTS_PER_PAGE-1 DO
			IF arrOutputFrameEmpty[iSelectedOutputPageIndex][iLoop] = FALSE THEN
				arrOutputFrame[iSelectedOutputPageIndex][iLoop].btnOut := arrOutputLink[iSelectedOutputPageIndex][iLoop].Out;
				
				IF arrOutputFrameEmpty[iSelectedOutputPageIndex][iLoop +1 ] = TRUE THEN
					EXIT;
					
				END_IF
			END_IF
		END_FOR
	END_IF
ELSIF ifUniversalMachineLink.State = MACHINE_STATE_EMERGENCY THEN
	eCurrentScreen := SCREEN_EMERGENCY;
	
END_IF
END_METHOD

METHOD PROTECTED ABSTRACT MS_Emergency
END_METHOD

METHOD PROTECTED MS_Initializing
VAR_INPUT
END_VAR
eCurrentNavigation := NAVIGATION_INITIALIZING;

IF ifUniversalMachineLink.State = MACHINE_STATE_UNINITIALIZED THEN
	eCurrentScreen := SCREEN_UNINITIALIZED;
			
ELSIF ifUniversalMachineLink.State = MACHINE_STATE_READY_INITIALIZED THEN
	eCurrentScreen := SCREEN_READY_INITIALIZED;
	
ELSIF ifUniversalMachineLink.State = MACHINE_STATE_AUTO THEN
	eCurrentScreen := SCREEN_AUTO;
	
ELSIF ifUniversalMachineLink.State = MACHINE_STATE_EMERGENCY THEN
	eCurrentScreen := SCREEN_EMERGENCY;
			
END_IF
END_METHOD

METHOD PROTECTED MS_Manual
VAR_INPUT
END_VAR
eCurrentNavigation := NAVIGATION_MANUAL;

//IF ifUniversalMachineLink.State = MACHINE_STATE_UNINITIALIZED THEN
//	eCurrentScreen := SCREEN_UNINITIALIZED;	
	
//ELSIF ifUniversalMachineLink.State = MACHINE_STATE_MANUAL_TO_AUTO THEN
//	eCurrentScreen := SCREEN_MODE_CHANGE;
	
//ELSIF ifUniversalMachineLink.State = MACHINE_STATE_EMERGENCY THEN
//	eCurrentScreen := SCREEN_EMERGENCY;
	
//END_IF

IF btnManualCylinder THEN
	eCurrentScreen := SCREEN_MANUAL_CYLINDERS;

ELSIF btnManualAxis THEN
	eCurrentScreen := SCREEN_MANUAL_MOTORS;
	
ELSIF btnManualInputs THEN
	eCurrentScreen := SCREEN_MANUAL_INPUTS;
	
ELSIF btnManualOutputs THEN
	eCurrentScreen := SCREEN_MANUAL_OUTPUTS;
	
//ELSIF btnManualSafety THEN
//	eCurrentScreen := SCREEN_MANUAL_SAFETY;

ELSIF btnManualRobots THEN
	eCurrentScreen := SCREEN_MANUAL_ROBOTS;

ELSIF btnManualOthers THEN
	eCurrentScreen := SCREEN_MANUAL_OTHERS;
	
END_IF
END_METHOD

METHOD PROTECTED MS_ManualAxis
VAR_INPUT
END_VAR
(*Set current screen *)
eCurrentScreen := SCREEN_MANUAL_MOTORS;

(* Run common part of manual pages handling *)
MS_Manual();

IF arrAxisFrameEmpty[iAxisPageIndex][0] THEN
    iAxisPageIndex := iAxisPageIndex - 1;
END_IF

bNextInvisible := iSelectedAxisPageIndex = iAxisPageIndex;
bPreviousInvisible := iSelectedAxisPageIndex = 0;

(* Frames control *)
IF btnPrevious THEN
	btnPrevious := FALSE;
	iSelectedAxisPageIndex := iSelectedAxisPageIndex - 1;
ELSIF btnNext THEN
	btnNext := FALSE;
	iSelectedAxisPageIndex := iSelectedAxisPageIndex + 1;
END_IF

IF iAxisIndex > 0 THEN
	FOR iLoop := 0 TO iAXIS_PER_PAGE-1 DO
		IF arrAxisFrameEmpty[iSelectedAxisPageIndex][iLoop] = FALSE THEN
			(* Assign object status to frame*)
			arrAxisFrame[iSelectedAxisPageIndex][iLoop].bActive := arrAxisLink[iSelectedAxisPageIndex][iLoop].Active;
			arrAxisFrame[iSelectedAxisPageIndex][iLoop].bHomed := arrAxisLink[iSelectedAxisPageIndex][iLoop].IsHomed;
			arrAxisFrame[iSelectedAxisPageIndex][iLoop].bInPosition := arrAxisLink[iSelectedAxisPageIndex][iLoop].InPosition;
			arrAxisFrame[iSelectedAxisPageIndex][iLoop].bHalted := arrAxisLink[iSelectedAxisPageIndex][iLoop].Halted;
			arrAxisFrame[iSelectedAxisPageIndex][iLoop].bError := arrAxisLink[iSelectedAxisPageIndex][iLoop].Error;
			arrAxisFrame[iSelectedAxisPageIndex][iLoop].iErrorID := arrAxisLink[iSelectedAxisPageIndex][iLoop].ErrorID;
			arrAxisFrame[iSelectedAxisPageIndex][iLoop].eAxisState := arrAxisLink[iSelectedAxisPageIndex][iLoop].State;
			arrAxisFrame[iSelectedAxisPageIndex][iLoop].lrActualPosition := arrAxisLink[iSelectedAxisPageIndex][iLoop].ActualPosition;
			arrAxisFrame[iSelectedAxisPageIndex][iLoop].lrActualVelocity := arrAxisLink[iSelectedAxisPageIndex][iLoop].ActualVelocity;
			arrAxisFrame[iSelectedAxisPageIndex][iLoop].lrSetPosition := arrAxisLink[iSelectedAxisPageIndex][iLoop].SetpointPosition;
			arrAxisFrame[iSelectedAxisPageIndex][iLoop].lrSetVelocity := arrAxisLink[iSelectedAxisPageIndex][iLoop].SetpointVelocity;
			arrAxisFrame[iSelectedAxisPageIndex][iLoop].lrLagError := arrAxisLink[iSelectedAxisPageIndex][iLoop].LagError;
			arrAxisFrame[iSelectedAxisPageIndex][iLoop].sName := arrAxisLink[iSelectedAxisPageIndex][iLoop].Name;
			arrAxisFrame[iSelectedAxisPageIndex][iLoop].sUnit := arrAxisLink[iSelectedAxisPageIndex][iLoop].Unit;
			
			(* Assign parameters from frame to object *)
			arrAxisLink[iSelectedAxisPageIndex][iLoop].Override := arrAxisFrame[iSelectedAxisPageIndex][iLoop].lrOverride;
			arrAxisLink[iSelectedAxisPageIndex][iLoop].JogPosition := arrAxisFrame[iSelectedAxisPageIndex][iLoop].lrJogDistance;
			arrAxisLink[iSelectedAxisPageIndex][iLoop].JogVelocity := arrAxisFrame[iSelectedAxisPageIndex][iLoop].lrJogVelocity;
			arrAxisLink[iSelectedAxisPageIndex][iLoop].JogAcceleration := arrAxisFrame[iSelectedAxisPageIndex][iLoop].lrJogAcceleration;
			arrAxisLink[iSelectedAxisPageIndex][iLoop].JogDeceleration := arrAxisFrame[iSelectedAxisPageIndex][iLoop].lrJogDeceleartion;
			
			(* Bound jog mode frame selector to axis object jog mode *)
			CASE arrAxisFrame[iSelectedAxisPageIndex][iLoop].eJogMode OF
				VISU_AXIS_JOG_MODE_STANDARD_SLOW:
					arrAxisLink[iSelectedAxisPageIndex][iLoop].JogMode := E_JogMode.MC_JOGMODE_STANDARD_SLOW;
					
				VISU_AXIS_JOG_MODE_STANDARD_FAST:
					arrAxisLink[iSelectedAxisPageIndex][iLoop].JogMode := E_JogMode.MC_JOGMODE_STANDARD_FAST;
					
				VISU_AXIS_JOG_MODE_CONTINOUS:
					arrAxisLink[iSelectedAxisPageIndex][iLoop].JogMode := E_JogMode.MC_JOGMODE_CONTINOUS;
					
				VISU_AXIS_JOG_MODE_INCHING:
					arrAxisLink[iSelectedAxisPageIndex][iLoop].JogMode := E_JogMode.MC_JOGMODE_INCHING;
					
				VISU_AXIS_JOG_MODE_INCHING_MODULO:
					arrAxisLink[iSelectedAxisPageIndex][iLoop].JogMode := E_JogMode.MC_JOGMODE_INCHING_MODULO;
					
			END_CASE
			
			(* Manual object control via requests *)
			IF arrAxisFrame[iSelectedAxisPageIndex][iLoop].btnReset THEN
				arrAxisFrame[iSelectedAxisPageIndex][iLoop].btnReset := FALSE;
				arrAxisState[iSelectedAxisPageIndex][iLoop] := VISU_CTRL_AXIS_RESET;
				
			ELSIF arrAxisFrame[iSelectedAxisPageIndex][iLoop].btnHalt THEN
				arrAxisFrame[iSelectedAxisPageIndex][iLoop].btnHalt := FALSE;
				arrAxisState[iSelectedAxisPageIndex][iLoop] := VISU_CTRL_AXIS_HALT;
				
			END_IF
			
			CASE arrAxisState[iSelectedAxisPageIndex][iLoop] OF
				VISU_CTRL_AXIS_WAIT_FOR_CMD:
					IF arrAxisFrame[iSelectedAxisPageIndex][iLoop].btnInit THEN
						arrAxisFrame[iSelectedAxisPageIndex][iLoop].btnInit := FALSE;
						arrAxisState[iSelectedAxisPageIndex][iLoop] := VISU_CTRL_AXIS_INIT;
						
					ELSIF arrAxisFrame[iSelectedAxisPageIndex][iLoop].btnHome THEN
						arrAxisFrame[iSelectedAxisPageIndex][iLoop].btnHome := FALSE;
						arrAxisState[iSelectedAxisPageIndex][iLoop] := VISU_CTRL_AXIS_HOME;
						
					ELSIF arrAxisFrame[iSelectedAxisPageIndex][iLoop].btnJogPositive THEN
						arrAxisState[iSelectedAxisPageIndex][iLoop] := VISU_CTRL_AXIS_JOG_POSITIVE;
						
					ELSIF arrAxisFrame[iSelectedAxisPageIndex][iLoop].btnJogNegative THEN
						arrAxisState[iSelectedAxisPageIndex][iLoop] := VISU_CTRL_AXIS_JOG_NEGATIVE;
						
					ELSIF arrAxisFrame[iSelectedAxisPageIndex][iLoop].btnAbort THEN
						arrAxisFrame[iSelectedAxisPageIndex][iLoop].btnAbort := FALSE;
						arrAxisState[iSelectedAxisPageIndex][iLoop] := VISU_CTRL_AXIS_ABORT;
						
					END_IF
					
				VISU_CTRL_AXIS_INIT:
					arrAxisLink[iSelectedAxisPageIndex][iLoop].MR_Init();
					
					IF arrAxisLink[iSelectedAxisPageIndex][iLoop].Active THEN
						arrAxisState[iSelectedAxisPageIndex][iLoop] := VISU_CTRL_AXIS_WAIT_FOR_CMD;
					END_IF
				
				VISU_CTRL_AXIS_HOME:
					arrAxisLink[iSelectedAxisPageIndex][iLoop].MR_Home(0.0);
					
					IF arrAxisLink[iSelectedAxisPageIndex][iLoop].IsHomed THEN
						arrAxisState[iSelectedAxisPageIndex][iLoop] := VISU_CTRL_AXIS_WAIT_FOR_CMD;
					END_IF
				
				VISU_CTRL_AXIS_RESET:
					arrAxisLink[iSelectedAxisPageIndex][iLoop].MR_Reset();
					
					IF NOT arrAxisLink[iSelectedAxisPageIndex][iLoop].Error AND NOT arrAxisLink[iSelectedAxisPageIndex][iLoop].Busy THEN
						arrAxisState[iSelectedAxisPageIndex][iLoop] := VISU_CTRL_AXIS_WAIT_FOR_CMD;
					END_IF
				
				VISU_CTRL_AXIS_JOG_POSITIVE:
					arrAxisLink[iSelectedAxisPageIndex][iLoop].JogDirection := E_AxisJogDirection.AXIS_JOG_DIR_POSITIVE;													
					arrAxisLink[iSelectedAxisPageIndex][iLoop].MR_Jog(bJogActive := arrAxisFrame[iSelectedAxisPageIndex][iLoop].btnJogPositive);
					
					IF arrAxisLink[iSelectedAxisPageIndex][iLoop].JogDone THEN
						arrAxisState[iSelectedAxisPageIndex][iLoop] := VISU_CTRL_AXIS_WAIT_FOR_CMD;
					END_IF
				
				VISU_CTRL_AXIS_JOG_NEGATIVE:
					arrAxisLink[iSelectedAxisPageIndex][iLoop].JogDirection := E_AxisJogDirection.AXIS_JOG_DIR_NEGATIVE;														
					arrAxisLink[iSelectedAxisPageIndex][iLoop].MR_Jog(bJogActive := arrAxisFrame[iSelectedAxisPageIndex][iLoop].btnJogNegative);
										
					IF arrAxisLink[iSelectedAxisPageIndex][iLoop].JogDone THEN
						arrAxisState[iSelectedAxisPageIndex][iLoop] := VISU_CTRL_AXIS_WAIT_FOR_CMD;
					END_IF
				
				VISU_CTRL_AXIS_HALT:
					arrAxisLink[iSelectedAxisPageIndex][iLoop].MR_Halt();
					
					IF arrAxisLink[iSelectedAxisPageIndex][iLoop].Halted THEN
						arrAxisState[iSelectedAxisPageIndex][iLoop] := VISU_CTRL_AXIS_WAIT_FOR_CMD;
					END_IF	
				
				VISU_CTRL_AXIS_ABORT:
					arrAxisLink[iSelectedAxisPageIndex][iLoop].MR_Abort();
					
					IF NOT arrAxisLink[iSelectedAxisPageIndex][iLoop].Active THEN
						arrAxisState[iSelectedAxisPageIndex][iLoop] := VISU_CTRL_AXIS_WAIT_FOR_CMD;
					END_IF
				
			END_CASE
			
			(* Check if next frame is empty and exit loop *)
			IF arrAxisFrameEmpty[iSelectedAxisPageIndex][iLoop + 1] = TRUE THEN
				EXIT;
			END_IF
		END_IF
	END_FOR
END_IF
END_METHOD

METHOD PROTECTED MS_ManualCylinders
VAR_INPUT
END_VAR
eCurrentScreen := SCREEN_MANUAL_CYLINDERS;

MS_Manual();

IF arrCylinderFrameEmpty[iCylinderPageIndex][0] THEN
	iCylinderPageIndex := iCylinderPageIndex - 1;
END_IF

bNextInvisible := iSelectedCylinderPageIndex = iCylinderPageIndex;
bPreviousInvisible := iSelectedCylinderPageIndex = 0;

(* Frames control *)
IF btnPrevious THEN
	btnPrevious := FALSE;
	iSelectedCylinderPageIndex := iSelectedCylinderPageIndex - 1;
ELSIF btnNext THEN
	btnNext := FALSE;
	iSelectedCylinderPageIndex := iSelectedCylinderPageIndex + 1;
END_IF

IF iCylinderIndex > 0 THEN
	FOR iLoop := 0 TO iCYLINDERS_PER_PAGE-1 DO
		IF arrCylinderFrameEmpty[iSelectedCylinderPageIndex][iLoop] = FALSE THEN
			arrCylinderFrame[iSelectedCylinderPageIndex][iLoop].bSensorActive := arrCylinderLink[iSelectedCylinderPageIndex][iLoop].PositionActive;
			arrCylinderFrame[iSelectedCylinderPageIndex][iLoop].bSensorHome := arrCylinderLink[iSelectedCylinderPageIndex][iLoop].PositionHome;
			arrCylinderFrame[iSelectedCylinderPageIndex][iLoop].bPositionHold := arrCylinderLink[iSelectedCylinderPageIndex][iLoop].PositionHold;
			arrCylinderFrame[iSelectedCylinderPageIndex][iLoop].bError := arrCylinderLink[iSelectedCylinderPageIndex][iLoop].Error;
			arrCylinderFrame[iSelectedCylinderPageIndex][iLoop].iErrorID := arrCylinderLink[iSelectedCylinderPageIndex][iLoop].ErrorID;
			arrCylinderFrame[iSelectedCylinderPageIndex][iLoop].eCylinderState := arrCylinderLink[iSelectedCylinderPageIndex][iLoop].State;
			arrCylinderFrame[iSelectedCylinderPageIndex][iLoop].sName := arrCylinderLink[iSelectedCylinderPageIndex][iLoop].Name;
			arrCylinderFrame[iSelectedCylinderPageIndex][iLoop].tActiveMovement := arrCylinderLink[iSelectedCylinderPageIndex][iLoop].MoveActiveTime;
			arrCylinderFrame[iSelectedCylinderPageIndex][iLoop].tHomeMovement := arrCylinderLink[iSelectedCylinderPageIndex][iLoop].MoveHomeTime;
			
			(* Requests handling *)
			IF arrCylinderFrame[iSelectedCylinderPageIndex][iLoop].btnReset THEN
				arrCylinderState[iSelectedCylinderPageIndex][iLoop] := VISU_CTRL_CYLINDER_RESET;
			END_IF
			
			CASE arrCylinderState[iSelectedCylinderPageIndex][iLoop] OF
				VISU_CTRL_CYLINDER_WAIT_FOR_CMD:
					IF arrCylinderFrame[iSelectedCylinderPageIndex][iLoop].btnInit THEN
						arrCylinderState[iSelectedCylinderPageIndex][iLoop] := VISU_CTRL_CYLINDER_INIT;
						
					ELSIF arrCylinderFrame[iSelectedCylinderPageIndex][iLoop].btnGoHome THEN
						arrCylinderState[iSelectedCylinderPageIndex][iLoop] := VISU_CTRL_CYLINDER_GO_HOME;
						
					ELSIF arrCylinderFrame[iSelectedCylinderPageIndex][iLoop].btnGoActive THEN
						arrCylinderState[iSelectedCylinderPageIndex][iLoop] := VISU_CTRL_CYLINDER_GO_ACTIVE;
						
					ELSIF arrCylinderFrame[iSelectedCylinderPageIndex][iLoop].btnRealase THEN
						arrCylinderState[iSelectedCylinderPageIndex][iLoop] := VISU_CTRL_CYLINDER_GO_RELEASE;
						
					ELSIF arrCylinderFrame[iSelectedCylinderPageIndex][iLoop].btnAbort THEN
						arrCylinderState[iSelectedCylinderPageIndex][iLoop] := VISU_CTRL_CYLINDER_ABORT;
						
					END_IF
					
				VISU_CTRL_CYLINDER_INIT:
					arrCylinderLink[iSelectedCylinderPageIndex][iLoop].MR_Init();
					
					IF arrCylinderLink[iSelectedCylinderPageIndex][iLoop].Active THEN
						arrCylinderState[iSelectedCylinderPageIndex][iLoop] := VISU_CTRL_CYLINDER_WAIT_FOR_CMD;
					END_IF
					
				VISU_CTRL_CYLINDER_RESET:
					arrCylinderLink[iSelectedCylinderPageIndex][iLoop].MR_Reset();
					
					IF NOT arrCylinderLink[iSelectedCylinderPageIndex][iLoop].Error THEN
						arrCylinderState[iSelectedCylinderPageIndex][iLoop] := VISU_CTRL_CYLINDER_WAIT_FOR_CMD;
					END_IF
				
				VISU_CTRL_CYLINDER_GO_HOME:
					arrCylinderLink[iSelectedCylinderPageIndex][iLoop].MR_GoHome();
					arrCylinderFrame[iSelectedCylinderPageIndex][iLoop].sHomeDescription := arrCylinderFrame[iSelectedCylinderPageIndex][iLoop].sHomeDescription;
					
					IF arrCylinderLink[iSelectedCylinderPageIndex][iLoop].PositionHome AND NOT arrCylinderLink[iSelectedCylinderPageIndex][iLoop].Busy THEN
						arrCylinderState[iSelectedCylinderPageIndex][iLoop] := VISU_CTRL_CYLINDER_WAIT_FOR_CMD;
					END_IF
				
				VISU_CTRL_CYLINDER_GO_ACTIVE:
					arrCylinderLink[iSelectedCylinderPageIndex][iLoop].MR_GoActive();
					arrCylinderFrame[iSelectedCylinderPageIndex][iLoop].sActiveDescription := arrCylinderFrame[iSelectedCylinderPageIndex][iLoop].sActiveDescription;
					
					IF arrCylinderLink[iSelectedCylinderPageIndex][iLoop].PositionActive AND NOT arrCylinderLink[iSelectedCylinderPageIndex][iLoop].Busy THEN
						arrCylinderState[iSelectedCylinderPageIndex][iLoop] := VISU_CTRL_CYLINDER_WAIT_FOR_CMD;
					END_IF
				
				VISU_CTRL_CYLINDER_GO_RELEASE:
					arrCylinderLink[iSelectedCylinderPageIndex][iLoop].MR_Release();
					
					IF NOT arrCylinderLink[iSelectedCylinderPageIndex][iLoop].PositionHold THEN
						arrCylinderState[iSelectedCylinderPageIndex][iLoop] := VISU_CTRL_CYLINDER_WAIT_FOR_CMD;
					END_IF
					
				VISU_CTRL_CYLINDER_ABORT:
					arrCylinderLink[iSelectedCylinderPageIndex][iLoop].MR_Abort();
					
					IF NOT arrCylinderLink[iSelectedCylinderPageIndex][iLoop].Active THEN
						arrCylinderState[iSelectedCylinderPageIndex][iLoop] := VISU_CTRL_CYLINDER_WAIT_FOR_CMD;
					END_IF
				
			END_CASE
			(* Check if next frame is empty and exit loop *)
			IF arrCylinderFrameEmpty[iSelectedCylinderPageIndex][iLoop + 1] = TRUE THEN
				EXIT;
			END_IF
		END_IF
	END_FOR
END_IF
END_METHOD

METHOD PROTECTED MS_ManualInputs
VAR_INPUT
END_VAR
eCurrentScreen := SCREEN_MANUAL_INPUTS;

MS_Manual();

IF arrInputFrameEmpty[iInputPageIndex][0] THEN
	iInputPageIndex := iInputPageIndex - 1;
END_IF

bNextInvisible := iSelectedInputPageIndex = iInputPageIndex;
bPreviousInvisible := iSelectedInputPageIndex = 0;

(* Frames control *)
IF btnPrevious THEN
	btnPrevious := FALSE;
	iSelectedInputPageIndex := iSelectedInputPageIndex - 1;
ELSIF btnNext THEN
	btnNext := FALSE;
	iSelectedInputPageIndex := iSelectedInputPageIndex + 1;
END_IF

IF iInputIndex > 0 THEN
	FOR iLoop := 0 TO iINPUTS_PER_PAGE-1 DO
		IF arrInputFrameEmpty[iSelectedInputPageIndex][iLoop] = FALSE THEN
			arrInputFrame[iSelectedInputPageIndex][iLoop].sName := arrInputLink[iSelectedInputPageIndex][iLoop].Name;
			arrInputFrame[iSelectedInputPageIndex][iLoop].sModuleType := arrInputLink[iSelectedInputPageIndex][iLoop].ModuleType;
			arrInputFrame[iSelectedInputPageIndex][iLoop].sPortID := arrInputLink[iSelectedInputPageIndex][iLoop].PortID;
			arrInputFrame[iSelectedInputPageIndex][iLoop].bIn := arrInputLink[iSelectedInputPageIndex][iLoop].In;
			
			arrInputLink[iSelectedInputPageIndex][iLoop].EnableForce := NOT(arrInputFrame[iSelectedInputPageIndex][iLoop].bForceDisabled);
			
			IF arrInputFrame[iSelectedInputPageIndex][iLoop].bForceIn THEN
				arrInputLink[iSelectedInputPageIndex][iLoop].MR_SetForceValue();
			ELSE 
				arrInputLink[iSelectedInputPageIndex][iLoop].MR_ResetForceValue();
			END_IF
			
			IF arrInputFrameEmpty[iSelectedInputPageIndex][iLoop + 1] = TRUE THEN
				EXIT;
			END_IF
		END_IF
	END_FOR
END_IF
END_METHOD

METHOD PROTECTED MS_ManualOthers
VAR_INPUT
END_VAR
eCurrentScreen := SCREEN_MANUAL_OTHERS;

MS_Manual();
END_METHOD

METHOD PROTECTED MS_ManualOutputs
VAR_INPUT
END_VAR
eCurrentScreen := SCREEN_MANUAL_OUTPUTS;

MS_Manual();

IF arrOutputFrameEmpty[iOutputPageIndex][0] THEN
	iOutputPageIndex := iOutputPageIndex - 1;
END_IF

bNextInvisible := iSelectedOutputPageIndex = iOutputPageIndex;
bPreviousInvisible := iSelectedOutputPageIndex = 0;

(* Frames control *)
IF btnPrevious THEN
	btnPrevious := FALSE;
	iSelectedOutputPageIndex := iSelectedOutputPageIndex - 1;
ELSIF btnNext THEN
	btnNext := FALSE;
	iSelectedOutputPageIndex := iSelectedOutputPageIndex + 1;
END_IF

IF iOutputIndex > 0 THEN
	FOR iLoop := 0 TO iOUTPUTS_PER_PAGE-1 DO
		IF arrOutputFrameEmpty[iSelectedOutputPageIndex][iLoop] = FALSE THEN
			//arrOutputFrame[iSelectedOutputPageIndex][iLoop].bControlable := arrOutputLink[iSelectedOutputPageIndex][iLoop].;
			arrOutputFrame[iSelectedOutputPageIndex][iLoop].sName := arrOutputLink[iSelectedOutputPageIndex][iLoop].Name;
			arrOutputFrame[iSelectedOutputPageIndex][iLoop].sModuleType := arrOutputLink[iSelectedOutputPageIndex][iLoop].ModuleType;
			arrOutputFrame[iSelectedOutputPageIndex][iLoop].sPortID := arrOutputLink[iSelectedOutputPageIndex][iLoop].PortID;
			arrOutputFrame[iSelectedOutputPageIndex][iLoop].bOut := arrOutputLink[iSelectedOutputPageIndex][iLoop].Out;
			
			(* Controll output *)
			arrOutputLink[iSelectedOutputPageIndex][iLoop].Out := arrOutputFrame[iSelectedOutputPageIndex][iLoop].btnOut;
			IF arrOutputFrameEmpty[iSelectedOutputPageIndex][iLoop +1 ] = TRUE THEN
				EXIT;
			END_IF
		END_IF
	END_FOR
END_IF
END_METHOD

METHOD PROTECTED MS_ManualRobots
VAR_INPUT
END_VAR
eCurrentScreen := SCREEN_MANUAL_ROBOTS;

MS_Manual();

IF arrRobotFrameEmpty[iRobotPageIndex][0] THEN
	iRobotPageIndex := iRobotPageIndex - 1;
END_IF

bNextInvisible := iSelectedRobotPageIndex = iRobotPageIndex;
bPreviousInvisible := iSelectedRobotPageIndex = 0;



(* Frames control *)
IF btnPrevious THEN
	btnPrevious := FALSE;
	iSelectedRobotPageIndex := iSelectedRobotPageIndex - 1;
ELSIF btnNext THEN
	btnNext := FALSE;
	iSelectedRobotPageIndex := iSelectedRobotPageIndex + 1;
END_IF

IF iRobotIndex > 0 THEN
	FOR iLoop := 0 TO iROBOTS_PER_PAGE-1 DO
		IF arrRobotFrameEmpty[iSelectedRobotPageIndex][iLoop] = FALSE THEN
			arrRobotFrame[iSelectedRobotPageIndex][iLoop].bIsHomed := arrRobotLink[iSelectedRobotPageIndex][iLoop].IsHomed;
			arrRobotFrame[iSelectedRobotPageIndex][iLoop].bInit := arrRobotLink[iSelectedRobotPageIndex][iLoop].Active;			
			arrRobotFrame[iSelectedRobotPageIndex][iLoop].bError := arrRobotLink[iSelectedRobotPageIndex][iLoop].Error;
			arrRobotFrame[iSelectedRobotPageIndex][iLoop].sErrorDescription := arrRobotLink[iSelectedRobotPageIndex][iLoop].ErrorName;
			arrRobotFrame[iSelectedRobotPageIndex][iLoop].eRobotState := arrRobotLink[iSelectedRobotPageIndex][iLoop].State;
			arrRobotFrame[iSelectedRobotPageIndex][iLoop].sName := arrRobotLink[iSelectedRobotPageIndex][iLoop].Name;
			arrRobotFrame[iSelectedRobotPageIndex][iLoop].bServoOff := arrRobotLink[iSelectedRobotPageIndex][iLoop].ServoIsOff;
			arrRobotFrame[iSelectedRobotPageIndex][iLoop].bServoOn := arrRobotLink[iSelectedRobotPageIndex][iLoop].ServoIsOn;
			arrRobotFrame[iSelectedRobotPageIndex][iLoop].bPaused := arrRobotLink[iSelectedRobotPageIndex][iLoop].Pausing;
			arrRobotFrame[iSelectedRobotPageIndex][iLoop].bStopped := arrRobotLink[iSelectedRobotPageIndex][iLoop].ProgramStopped;
			arrRobotFrame[iSelectedRobotPageIndex][iLoop].bStarted := arrRobotLink[iSelectedRobotPageIndex][iLoop].DoingAction;
			arrRobotFrame[iSelectedRobotPageIndex][iLoop].bPowerOn := arrRobotLink[iSelectedRobotPageIndex][iLoop].CR800PoweredOn;			
			arrRobotFrame[iSelectedRobotPageIndex][iLoop].bBatteryLow := arrRobotLink[iSelectedRobotPageIndex][iLoop].BatteryLow;	
			arrRobotFrame[iSelectedRobotPageIndex][iLoop].bUninitialized := arrRobotLink[iSelectedRobotPageIndex][iLoop].Uninitialized;			
			
			(* Assign parameters from frame to object *)
			arrRobotLink[iSelectedRobotPageIndex][iLoop].ActionNumber := arrRobotFrame[iSelectedRobotPageIndex][iLoop].iActionNumber;
			arrRobotLink[iSelectedRobotPageIndex][iLoop].Override := arrRobotFrame[iSelectedRobotPageIndex][iLoop].iOverride;
			
			(* Assigning state of button disable *)
			arrRobotFrame[iSelectedRobotPageIndex][iLoop].bModeSwitchButtonDisabled := bModeSwitchButtonDisabled;
						
			IF arrRobotLink[iSelectedRobotPageIndex][iLoop].Uninitialized OR arrRobotLink[iSelectedRobotPageIndex][iLoop].AutoModeStarted OR NOT arrRobotLink[iSelectedRobotPageIndex][iLoop].IsHomed THEN
				arrRobotFrame[iSelectedRobotPageIndex][iLoop].bAutoButtonDisable := TRUE;
			ELSE
				arrRobotFrame[iSelectedRobotPageIndex][iLoop].bAutoButtonDisable := FALSE;
			END_IF

			IF arrRobotLink[iSelectedRobotPageIndex][iLoop].Uninitialized OR arrRobotLink[iSelectedRobotPageIndex][iLoop].IsHomed THEN
				arrRobotFrame[iSelectedRobotPageIndex][iLoop].bHomeButtonDisable := TRUE;
			ELSE
				arrRobotFrame[iSelectedRobotPageIndex][iLoop].bHomeButtonDisable := FALSE;
			END_IF
			
			IF arrRobotLink[iSelectedRobotPageIndex][iLoop].Uninitialized OR NOT arrRobotLink[iSelectedRobotPageIndex][iLoop].AutoModeStarted OR arrRobotLink[iSelectedRobotPageIndex][iLoop].DoingAction OR arrRobotLink[iSelectedRobotPageIndex][iLoop].Pausing OR arrRobotLink[iSelectedRobotPageIndex][iLoop].ProgramStopped THEN
				arrRobotFrame[iSelectedRobotPageIndex][iLoop].bActionButtonDisable := TRUE;
			ELSE
				arrRobotFrame[iSelectedRobotPageIndex][iLoop].bActionButtonDisable := FALSE;
			END_IF

			IF arrRobotLink[iSelectedRobotPageIndex][iLoop].Uninitialized OR NOT arrRobotLink[iSelectedRobotPageIndex][iLoop].DoingAction OR arrRobotLink[iSelectedRobotPageIndex][iLoop].Pausing OR arrRobotLink[iSelectedRobotPageIndex][iLoop].ProgramStopped THEN
				arrRobotFrame[iSelectedRobotPageIndex][iLoop].bPausingButtonDisable := TRUE;
			ELSE
				arrRobotFrame[iSelectedRobotPageIndex][iLoop].bPausingButtonDisable := FALSE;
			END_IF
			
			IF arrRobotLink[iSelectedRobotPageIndex][iLoop].Uninitialized OR NOT arrRobotLink[iSelectedRobotPageIndex][iLoop].Pausing OR arrRobotLink[iSelectedRobotPageIndex][iLoop].ProgramStopped THEN
				arrRobotFrame[iSelectedRobotPageIndex][iLoop].bRestoreCycleButtonDisable := TRUE;
			ELSE
				arrRobotFrame[iSelectedRobotPageIndex][iLoop].bRestoreCycleButtonDisable := FALSE;
			END_IF	

			IF arrRobotLink[iSelectedRobotPageIndex][iLoop].Uninitialized OR NOT arrRobotLink[iSelectedRobotPageIndex][iLoop].DoingAction OR arrRobotLink[iSelectedRobotPageIndex][iLoop].ProgramStopped OR arrRobotLink[iSelectedRobotPageIndex][iLoop].Pausing THEN
				arrRobotFrame[iSelectedRobotPageIndex][iLoop].bStoppingButtonDisable := TRUE;
			ELSE
				arrRobotFrame[iSelectedRobotPageIndex][iLoop].bStoppingButtonDisable := FALSE;
			END_IF	
			
			IF arrRobotLink[iSelectedRobotPageIndex][iLoop].Uninitialized OR NOT arrRobotLink[iSelectedRobotPageIndex][iLoop].ProgramStopped OR arrRobotLink[iSelectedRobotPageIndex][iLoop].Pausing THEN
				arrRobotFrame[iSelectedRobotPageIndex][iLoop].bRestoreAutoButtonDisable := TRUE;
			ELSE
				arrRobotFrame[iSelectedRobotPageIndex][iLoop].bRestoreAutoButtonDisable := FALSE;
			END_IF	
		
			(* Requests handling *)
			IF arrRobotFrame[iSelectedRobotPageIndex][iLoop].btnErrorReset THEN
				arrRobotState[iSelectedRobotPageIndex][iLoop] := VISU_CTRL_ROBOT_ERR_RESET;
			END_IF
			
			(* Requests handling *)
			IF arrRobotFrame[iSelectedRobotPageIndex][iLoop].btnControllerReset THEN
				arrRobotState[iSelectedRobotPageIndex][iLoop] := VISU_CTRL_ROBOT_CONTROLLER_RESET;
			END_IF
			
			(* Requests handling *)
			IF arrRobotFrame[iSelectedRobotPageIndex][iLoop].btnAbort THEN
				arrRobotState[iSelectedRobotPageIndex][iLoop] := VISU_CTRL_ROBOT_ABORT;
			END_IF
			
			IF arrRobotFrame[iSelectedRobotPageIndex][iLoop].btnCyclePause THEN
				arrRobotState[iSelectedRobotPageIndex][iLoop] := VISU_CTRL_ROBOT_CYCLE_PAUSE;
			END_IF			
			
			IF arrRobotFrame[iSelectedRobotPageIndex][iLoop].btnCycleStop THEN
				arrRobotState[iSelectedRobotPageIndex][iLoop] := VISU_CTRL_ROBOT_CYCLE_STOP;
			END_IF	
	
			CASE arrRobotState[iSelectedRobotPageIndex][iLoop] OF
				VISU_CTRL_ROBOT_WAIT_FOR_CMD:
					IF arrRobotFrame[iSelectedRobotPageIndex][iLoop].btnInit THEN
						arrRobotState[iSelectedRobotPageIndex][iLoop] := VISU_CTRL_ROBOT_INIT;
						
					ELSIF arrRobotFrame[iSelectedRobotPageIndex][iLoop].btnGoHome THEN
						arrRobotState[iSelectedRobotPageIndex][iLoop] := VISU_CTRL_ROBOT_GO_HOME;
						
					ELSIF arrRobotFrame[iSelectedRobotPageIndex][iLoop].btnDoAction THEN
						arrRobotState[iSelectedRobotPageIndex][iLoop] := VISU_CTRL_ROBOT_DO_ACTION;
						
					ELSIF arrRobotFrame[iSelectedRobotPageIndex][iLoop].btnUpdateRecipes THEN
						arrRobotState[iSelectedRobotPageIndex][iLoop] := VISU_CTRL_ROBOT_UPDATE_RECIPES;
						
					ELSIF arrRobotFrame[iSelectedRobotPageIndex][iLoop].btnGoAuto THEN
						arrRobotState[iSelectedRobotPageIndex][iLoop] := VISU_CTRL_ROBOT_GO_AUTO;
						
					ELSIF arrRobotFrame[iSelectedRobotPageIndex][iLoop].btnRestoreCycle THEN
						arrRobotState[iSelectedRobotPageIndex][iLoop] := VISU_CTRL_ROBOT_RESTORE_CYCLE;
						
					ELSIF arrRobotFrame[iSelectedRobotPageIndex][iLoop].btnRestoreAuto THEN
						arrRobotState[iSelectedRobotPageIndex][iLoop] := VISU_CTRL_ROBOT_RESTORE_AUTO;

					ELSIF arrRobotFrame[iSelectedRobotPageIndex][iLoop].btnBatteryReset THEN
						arrRobotState[iSelectedRobotPageIndex][iLoop] := VISU_CTRL_ROBOT_BATTERY_RESET;
						
					END_IF

					
				VISU_CTRL_ROBOT_INIT:
					arrRobotLink[iSelectedRobotPageIndex][iLoop].MR_Init();
					
					IF arrRobotLink[iSelectedRobotPageIndex][iLoop].Active THEN
						arrRobotState[iSelectedRobotPageIndex][iLoop] := VISU_CTRL_ROBOT_WAIT_FOR_CMD;
					END_IF
					
				VISU_CTRL_ROBOT_ERR_RESET:
					arrRobotLink[iSelectedRobotPageIndex][iLoop].MR_Reset();
					
					IF NOT arrRobotLink[iSelectedRobotPageIndex][iLoop].Busy THEN
						arrRobotState[iSelectedRobotPageIndex][iLoop] := VISU_CTRL_ROBOT_WAIT_FOR_CMD;
					END_IF
				
				VISU_CTRL_ROBOT_CONTROLLER_RESET:
					arrRobotLink[iSelectedRobotPageIndex][iLoop].MR_ResetCR800Err();
					
					IF NOT arrRobotLink[iSelectedRobotPageIndex][iLoop].Busy THEN
						arrRobotState[iSelectedRobotPageIndex][iLoop] := VISU_CTRL_ROBOT_WAIT_FOR_CMD;
					END_IF
				
				VISU_CTRL_ROBOT_ABORT:
					arrRobotLink[iSelectedRobotPageIndex][iLoop].MR_Abort();
					
					IF NOT arrRobotLink[iSelectedRobotPageIndex][iLoop].Active THEN
						arrRobotState[iSelectedRobotPageIndex][iLoop] := VISU_CTRL_ROBOT_WAIT_FOR_CMD;
					END_IF
				
				VISU_CTRL_ROBOT_GO_HOME:
					arrRobotLink[iSelectedRobotPageIndex][iLoop].MR_GoHome();
					
					IF NOT arrRobotLink[iSelectedRobotPageIndex][iLoop].Busy THEN
						arrRobotState[iSelectedRobotPageIndex][iLoop] := VISU_CTRL_ROBOT_WAIT_FOR_CMD;
					END_IF
					
				VISU_CTRL_ROBOT_DO_ACTION:
					arrRobotLink[iSelectedRobotPageIndex][iLoop].MR_DoAction(arrRobotFrame[iSelectedRobotPageIndex][iLoop].iActionNumber);
					
					IF NOT arrRobotLink[iSelectedRobotPageIndex][iLoop].Busy THEN
						arrRobotState[iSelectedRobotPageIndex][iLoop] := VISU_CTRL_ROBOT_WAIT_FOR_CMD;
					END_IF

				VISU_CTRL_ROBOT_UPDATE_RECIPES:
					arrRobotLink[iSelectedRobotPageIndex][iLoop].MR_UpdateRecipies();
					
					IF NOT arrRobotLink[iSelectedRobotPageIndex][iLoop].Busy THEN
						arrRobotState[iSelectedRobotPageIndex][iLoop] := VISU_CTRL_ROBOT_WAIT_FOR_CMD;
					END_IF
			
				VISU_CTRL_ROBOT_GO_AUTO:
					arrRobotLink[iSelectedRobotPageIndex][iLoop].MR_GoAuto();
					
					IF NOT arrRobotLink[iSelectedRobotPageIndex][iLoop].Busy THEN
						arrRobotState[iSelectedRobotPageIndex][iLoop] := VISU_CTRL_ROBOT_WAIT_FOR_CMD;
					END_IF

				VISU_CTRL_ROBOT_CYCLE_PAUSE:
					arrRobotLink[iSelectedRobotPageIndex][iLoop].MR_CyclePause();
					
					IF NOT arrRobotLink[iSelectedRobotPageIndex][iLoop].Busy THEN
						arrRobotState[iSelectedRobotPageIndex][iLoop] := VISU_CTRL_ROBOT_WAIT_FOR_CMD;
					END_IF

				VISU_CTRL_ROBOT_CYCLE_STOP:
					arrRobotLink[iSelectedRobotPageIndex][iLoop].MR_CycleStop();
					
					IF NOT arrRobotLink[iSelectedRobotPageIndex][iLoop].Busy THEN
						arrRobotState[iSelectedRobotPageIndex][iLoop] := VISU_CTRL_ROBOT_WAIT_FOR_CMD;
					END_IF

				VISU_CTRL_ROBOT_RESTORE_CYCLE:
					arrRobotLink[iSelectedRobotPageIndex][iLoop].MR_RestoreCycle();
					
					IF NOT arrRobotLink[iSelectedRobotPageIndex][iLoop].Busy THEN
						arrRobotState[iSelectedRobotPageIndex][iLoop] := VISU_CTRL_ROBOT_WAIT_FOR_CMD;
					END_IF

				VISU_CTRL_ROBOT_RESTORE_AUTO:
					arrRobotLink[iSelectedRobotPageIndex][iLoop].MR_RestoreAuto();
					
					IF NOT arrRobotLink[iSelectedRobotPageIndex][iLoop].Busy THEN
						arrRobotState[iSelectedRobotPageIndex][iLoop] := VISU_CTRL_ROBOT_WAIT_FOR_CMD;
					END_IF
					
				VISU_CTRL_ROBOT_BATTERY_RESET:
					arrRobotLink[iSelectedRobotPageIndex][iLoop].MR_BatteryReset();
					
					IF NOT arrRobotLink[iSelectedRobotPageIndex][iLoop].Busy THEN
						arrRobotState[iSelectedRobotPageIndex][iLoop] := VISU_CTRL_ROBOT_WAIT_FOR_CMD;
					END_IF		
					
			END_CASE
			(* Check if next frame is empty and exit loop *)
			IF arrRobotFrameEmpty[iSelectedRobotPageIndex][iLoop + 1] = TRUE THEN
				EXIT;
			END_IF
		END_IF
	END_FOR
END_IF
END_METHOD

METHOD PROTECTED MS_ManualSafety
VAR_INPUT
END_VAR
eCurrentScreen := SCREEN_MANUAL_SAFETY;

MS_Manual();

IF arrSafeInputFrameEmpty[iSafeInputPageIndex][0] THEN
	iSafeInputPageIndex := iSafeInputPageIndex - 1;
END_IF

bNextInvisibleInput := iSelectedSafeInputPageIndex = iSafeInputPageIndex;
bPreviousInvisibleInput := iSelectedSafeInputPageIndex = 0;

(* Frames control *)
IF btnPreviousInput THEN
	btnPreviousInput := FALSE;
	iSelectedSafeInputPageIndex := iSelectedSafeInputPageIndex - 1;
ELSIF btnNextInput THEN
	btnNextInput := FALSE;
	iSelectedSafeInputPageIndex := iSelectedSafeInputPageIndex + 1;
END_IF

IF iSafeInputIndex > 0 THEN
	FOR iLoop := 0 TO iSAFE_INPUTS_PER_PAGE-1 DO
		IF arrSafeInputFrameEmpty[iSelectedSafeInputPageIndex][iLoop] = FALSE THEN
			arrSafeInputFrame[iSelectedSafeInputPageIndex][iLoop].sName := arrSafeInputLink[iSelectedSafeInputPageIndex][iLoop].Name;
			arrSafeInputFrame[iSelectedSafeInputPageIndex][iLoop].sModuleType := arrSafeInputLink[iSelectedSafeInputPageIndex][iLoop].ModuleType;
			arrSafeInputFrame[iSelectedSafeInputPageIndex][iLoop].sPortID := arrSafeInputLink[iSelectedSafeInputPageIndex][iLoop].PortID;
			arrSafeInputFrame[iSelectedSafeInputPageIndex][iLoop].bIn := arrSafeInputLink[iSelectedSafeInputPageIndex][iLoop].In;
			
			arrSafeInputLink[iSelectedSafeInputPageIndex][iLoop].EnableForce := NOT(arrSafeInputFrame[iSelectedSafeInputPageIndex][iLoop].bForceDisabled);
			
			IF arrSafeInputFrame[iSelectedSafeInputPageIndex][iLoop].bForceIn THEN
				arrSafeInputLink[iSelectedSafeInputPageIndex][iLoop].MR_SetForceValue();
			ELSE 
				arrSafeInputLink[iSelectedSafeInputPageIndex][iLoop].MR_ResetForceValue();
			END_IF
			
			IF arrSafeInputFrameEmpty[iSelectedSafeInputPageIndex][iLoop + 1] = TRUE THEN
				EXIT;
			END_IF
		END_IF
	END_FOR
END_IF

IF arrSafeOutputFrameEmpty[iSafeOutputPageIndex][0] THEN
	iSafeOutputPageIndex := iSafeOutputPageIndex - 1;
END_IF

bNextInvisibleOutput := iSelectedSafeOutputPageIndex = iSafeOutputPageIndex;
bPreviousInvisibleOutput := iSelectedSafeOutputPageIndex = 0;

(* Frames control *)
IF btnPreviousOutput THEN
	btnPreviousOutput := FALSE;
	iSelectedSafeOutputPageIndex := iSelectedSafeOutputPageIndex - 1;
ELSIF btnNextOutput THEN
	btnNextOutput := FALSE;
	iSelectedSafeOutputPageIndex := iSelectedSafeOutputPageIndex + 1;
END_IF


IF iSafeOutputIndex > 0 THEN
	FOR iLoop := 0 TO iSAFE_OUTPUTS_PER_PAGE-1 DO
		IF arrSafeOutputFrameEmpty[iSelectedOutputPageIndex][iLoop] = FALSE THEN
			//arrOutputFrame[iSelectedOutputPageIndex][iLoop].bControlable := arrOutputLink[iSelectedOutputPageIndex][iLoop].;
			arrSafeOutputFrame[iSelectedSafeOutputPageIndex][iLoop].sName := arrSafeOutputLink[iSelectedSafeOutputPageIndex][iLoop].Name;
			arrSafeOutputFrame[iSelectedSafeOutputPageIndex][iLoop].sModuleType := arrSafeOutputLink[iSelectedSafeOutputPageIndex][iLoop].ModuleType;
			arrSafeOutputFrame[iSelectedSafeOutputPageIndex][iLoop].sPortID := arrSafeOutputLink[iSelectedSafeOutputPageIndex][iLoop].PortID;
			arrSafeOutputFrame[iSelectedSafeOutputPageIndex][iLoop].bOut := arrSafeOutputLink[iSelectedSafeOutputPageIndex][iLoop].Out;
			
			(* Controll output *)
			arrSafeOutputLink[iSelectedSafeOutputPageIndex][iLoop].Out := arrSafeOutputFrame[iSelectedSafeOutputPageIndex][iLoop].btnOut;
			IF arrSafeOutputFrameEmpty[iSelectedSafeOutputPageIndex][iLoop +1 ] = TRUE THEN
				EXIT;
			END_IF
		END_IF
	END_FOR
END_IF
END_METHOD

METHOD PROTECTED MS_ModeChange
VAR_INPUT
END_VAR
eCurrentNavigation := NAVIGATION_EMPTY;

IF ifUniversalMachineLink.State = MACHINE_STATE_AUTO THEN
	eCurrentScreen := SCREEN_AUTO;	
	
ELSIF ifUniversalMachineLink.State = MACHINE_STATE_MANUAL THEN	
	eCurrentScreen := SCREEN_MANUAL_CYLINDERS;
	
ELSIF ifUniversalMachineLink.State = MACHINE_STATE_EMERGENCY THEN
	eCurrentScreen := SCREEN_EMERGENCY;
	
END_IF
END_METHOD

METHOD PROTECTED MS_ReadyInitialized
VAR_INPUT
END_VAR
eCurrentNavigation := NAVIGATION_INITIALIZING;

IF ifUniversalMachineLink.State = MACHINE_STATE_ABORTING THEN
	eCurrentScreen := SCREEN_ABORTING;	
			
ELSIF ifUniversalMachineLink.State = MACHINE_STATE_AUTO THEN
	eCurrentScreen := SCREEN_AUTO;
	
ELSIF ifUniversalMachineLink.State = MACHINE_STATE_EMERGENCY THEN
	eCurrentScreen := SCREEN_EMERGENCY;
			
END_IF
END_METHOD

METHOD PROTECTED MS_Recipes
VAR_INPUT
END_VAR
eCurrentNavigation := NAVIGATION_UTILITIES;

IF btnBack THEN
	btnBack := FALSE;
	eCurrentScreen := eLastScreen;
	
END_IF

IF arrRobotFrameEmpty[iRecipeParameterPageIndex][0] THEN
	iRecipeParameterPageIndex := iRecipeParameterPageIndex - 1;
END_IF

bRecipeNextInvisible := iSelectedRecipeParameterPageIndex = iRecipeParameterPageIndex;
bRecipePreviousInvisible := iSelectedRecipeParameterPageIndex = 0;

(* Frames control *)
IF btnPrevious THEN
	btnPrevious := FALSE;
	iSelectedRecipeParameterPageIndex := iSelectedRecipeParameterPageIndex - 1;
	
ELSIF btnNext THEN
	btnNext := FALSE;
	iSelectedRecipeParameterPageIndex := iSelectedRecipeParameterPageIndex + 1;
	
END_IF
END_METHOD

METHOD PROTECTED MS_Reset
VAR_INPUT
END_VAR
eCurrentNavigation := NAVIGATION_INITIALIZING;

IF ifUniversalMachineLink.State = MACHINE_STATE_RESET THEN
	eCurrentScreen := SCREEN_RESET;
	
ELSIF ifUniversalMachineLink.State = MACHINE_STATE_RESET_DONE THEN
	eCurrentScreen := SCREEN_AUTO;
	
ELSIF ifUniversalMachineLink.State = MACHINE_STATE_EMERGENCY THEN
	eCurrentScreen := SCREEN_EMERGENCY;
	
END_IF
END_METHOD

METHOD PROTECTED MS_Uninitialized
VAR_INPUT
END_VAR
eCurrentNavigation := NAVIGATION_UNINITIALIZED;
MS_Manual();
IF ifUniversalMachineLink.State = MACHINE_STATE_INITIALIZING THEN
	eCurrentScreen := SCREEN_INITIALIZING;	
	
END_IF
END_METHOD

PROPERTY Start : REFERENCE TO BOOL
GET
Start REF= btnStart;
END_GET
END_PROPERTY

METHOD PROTECTED StateMachine
VAR_INPUT
END_VAR
CASE eCurrentScreen OF
	SCREEN_UNINITIALIZED:
		MS_Uninitialized();
	
	SCREEN_INITIALIZING:
		MS_Initializing();
		
	SCREEN_READY_INITIALIZED:
		MS_ReadyInitialized();
		
	SCREEN_AUTO:
		MS_Auto();
		
	SCREEN_MODE_CHANGE:
		MS_ModeChange();
	
	SCREEN_MANUAL_CYLINDERS:
		MS_ManualCylinders();
		
	SCREEN_MANUAL_MOTORS:
		MS_ManualAxis();
	
//	SCREEN_MANUAL_SAFETY:
//		MS_ManualSafety();
	
	SCREEN_MANUAL_INPUTS:
		MS_ManualInputs();
	
	SCREEN_MANUAL_OUTPUTS:
		MS_ManualOutputs();
		
	SCREEN_MANUAL_ROBOTS:
		MS_ManualRobots();		
		
	SCREEN_MANUAL_OTHERS:
		MS_ManualOthers();
	
	SCREEN_ALARMS:
		MS_Alarms();
	
	SCREEN_RECIPES:
		MS_Recipes();
		
	SCREEN_RESET:
		MS_Reset();
		
	SCREEN_ABORTING:
		MS_Aborting();
		
	SCREEN_EMERGENCY:
		MS_Emergency();
	
END_CASE
END_METHOD

PROPERTY Stop : REFERENCE TO BOOL
GET
Stop REF= btnStop;
END_GET
END_PROPERTY

END_FUNCTION_BLOCK

// ---- POUs/Libs/Utilities/Systemtime to String/FUN_TimestructToDate.TcPOU
FUNCTION FUN_TimestructToDate : STRING
VAR_INPUT
	stTime : TIMESTRUCT;
END_VAR
VAR
	sTime : STRING;
END_VAR

sTime := SYSTEMTIME_TO_STRING(stTime);
FUN_TimestructToDate := LEFT(sTime,10);

END_FUNCTION

// ---- POUs/Libs/Utilities/Systemtime to String/FUN_TimestructToTime.TcPOU
FUNCTION FUN_TimestructToTime : STRING
VAR_INPUT
	stTime : TIMESTRUCT;
END_VAR
VAR
	sTime : STRING;
END_VAR

sTime := SYSTEMTIME_TO_STRING(stTime);
FUN_TimestructToTime := RIGHT(sTime,12);

END_FUNCTION

// ---- POUs/Libs/0_Checks/Checks/CheckBounds.TcPOU
// Implicitly generated code : DO NOT EDIT
FUNCTION CheckBounds : DINT
VAR_INPUT
	index, lower, upper: DINT;
END_VAR

// Implicitly generated code : Only an Implementation suggestion
IF  index < lower THEN
	CheckBounds := lower;
	GVL_Checks.dCheckBounds := GVL_Checks.dCheckBounds + 1;
//	ADSLOGSTR(4,'Checks critical error - index out of range','');
ELSIF  index > upper THEN
	CheckBounds := upper;
	GVL_Checks.dCheckBounds := GVL_Checks.dCheckBounds + 1;
//	ADSLOGSTR(4,'Checks critical error - index out of range','');
ELSE  
	CheckBounds := index;
END_IF

END_FUNCTION

// ---- POUs/Libs/0_Checks/Checks/CheckDivDInt.TcPOU
// Implicitly generated code : DO NOT EDIT
FUNCTION CheckDivDInt : DINT
VAR_INPUT
	divisor:DINT;
END_VAR

// Implicitly generated code : Only an Implementation suggestion
IF divisor = 0 THEN
	CheckDivDInt:=1;
	GVL_Checks.dCheckDivDInt := GVL_Checks.dCheckDivDInt + 1;
	ADSLOGSTR(4,'Checks critical error - DINT variable divided by 0.','');
ELSE
	CheckDivDInt:=divisor;
END_IF

END_FUNCTION

// ---- POUs/Libs/0_Checks/Checks/CheckDivLInt.TcPOU
// Implicitly generated code : DO NOT EDIT
FUNCTION CheckDivLInt : LINT
VAR_INPUT
	divisor:LINT;
END_VAR

// Implicitly generated code : Only an Implementation suggestion
IF divisor = 0 THEN
	CheckDivLInt:=1;
	GVL_Checks.dCheckDivLInt := GVL_Checks.dCheckDivLInt + 1;
	ADSLOGSTR(4,'Checks critical error - LINT variable divided by 0.','');
ELSE
	CheckDivLInt:=divisor;
END_IF

END_FUNCTION

// ---- POUs/Libs/0_Checks/Checks/CheckDivLReal.TcPOU
// Implicitly generated code : DO NOT EDIT
FUNCTION CheckDivLReal : LREAL
VAR_INPUT
	divisor:LREAL;
END_VAR

// Implicitly generated code : Only an Implementation suggestion
IF divisor = 0 THEN
	CheckDivLReal:=1;
	GVL_Checks.dCheckDivLReal := GVL_Checks.dCheckDivLReal + 1;
	ADSLOGSTR(4,'Checks critical error - DINT variable divided by 0.','');
ELSE
	CheckDivLReal:=divisor;
END_IF

END_FUNCTION

// ---- POUs/Libs/0_Checks/Checks/CheckDivReal.TcPOU
// Implicitly generated code : DO NOT EDIT
FUNCTION CheckDivReal : REAL
VAR_INPUT
	divisor:REAL;
END_VAR

// Implicitly generated code : Only an Implementation suggestion
IF divisor = 0 THEN
	CheckDivReal:=1;
	GVL_Checks.dCheckDivReal := GVL_Checks.dCheckDivReal + 1;
	ADSLOGSTR(4,'Checks critical error - DINT variable divided by 0.','');
ELSE
	CheckDivReal:=divisor;
END_IF

END_FUNCTION

// ---- POUs/Libs/0_Checks/Checks/CheckPointer.TcPOU
// Implicitly generated code : DO NOT EDIT
FUNCTION CheckPointer : POINTER TO BYTE
VAR_INPUT 
	ptToTest : POINTER TO BYTE; // Destination address of the pointer
	iSize : DINT;		        // Size of the type the pointer points to. (e.g: 20 for POINTER TO ARRAY [0..9] OF INT) 
	iGran : DINT;		        // Granularity of the pointer access. This is the size of the biggest non-structured data type in the type the pointer points to. (e.g: 2 for POINTER TO ARRAY [0..9] OF INT)
	bWrite: BOOL;		        // Indicates read or write Access. TRUE = write access.
END_VAR

// No standard way of implementation. Fill your own code here
CheckPointer := ptToTest;

END_FUNCTION

// ---- POUs/Libs/0_Checks/Checks/CheckRangeSigned.TcPOU
// Implicitly generated code : DO NOT EDIT
FUNCTION CheckRangeSigned : DINT
VAR_INPUT
	value, lower, upper: DINT;
END_VAR

// Implicitly generated code : Only an Implementation suggestion
IF (value < lower) THEN
	CheckRangeSigned := lower;
	GVL_Checks.dCheckRangeSigned := GVL_Checks.dCheckRangeSigned + 1;
	ADSLOGSTR(4,'Checks critical error - DINT overflow.','');
ELSIF(value > upper) THEN
	CheckRangeSigned := upper;
	GVL_Checks.dCheckRangeSigned := GVL_Checks.dCheckRangeSigned + 1;
	ADSLOGSTR(4,'Checks critical error - DINT overflow.','');
ELSE
	CheckRangeSigned := value;
END_IF

END_FUNCTION

// ---- POUs/Libs/0_Checks/Checks/CheckRangeUnsigned.TcPOU
// Implicitly generated code : DO NOT EDIT
FUNCTION CheckRangeUnsigned : UDINT
VAR_INPUT
	value, lower, upper: UDINT;
END_VAR

// Implicitly generated code : Only an Implementation suggestion
IF (value < lower) THEN
	CheckRangeUnsigned := lower;
	GVL_Checks.dCheckRangeUnsigned := GVL_Checks.dCheckRangeUnsigned + 1;
	ADSLOGSTR(4,'Checks critical error - UDINT overflow.','');
ELSIF(value > upper) THEN
	CheckRangeUnsigned := upper;
	GVL_Checks.dCheckRangeUnsigned := GVL_Checks.dCheckRangeUnsigned + 1;
	ADSLOGSTR(4,'Checks critical error - UDINT overflow.','');
ELSE
	CheckRangeUnsigned := value;
END_IF

END_FUNCTION

// ---- POUs/Libs/0_Checks/Checks/P_Checks.TcPOU
//==================================================================================================
//							Beckhoff Automation Poland
//									19.10.2018
//	Program wykrywajacy bledy dzielnia przez 0 i przekraczania zakresow zmiennych, tablic...
// 
//	v1.4	|| TC v 3.1.4022.25		|| - Ustawiono setowanie bledow, dodano wejscie bReset 
//	v1.3	|| TC v 3.1.4022.16		|| - Przeniesiono logowanie do EventLoggera wraz z zabepieczeniem przed zbyt szybkim logowaniem zdarzeń do programu P_SystemDiag_EventLog. 
//	v1.2	|| TC v 3.1.4020.28		|| - Dodano logowanie do EventLoggera wraz z zabepieczeniem przed zbyt szybki logowaniem zdarzeń
//	v1.1 	|| TC v 3.1.4020.14 	|| - Dodane wyjscia bOk, bWarning, bError
//	v1.0 	|| TC v 3.1.4020.0 		|| - Pierwsza wersja
//==================================================================================================
PROGRAM P_Checks
VAR_INPUT
	bReset							: BOOL;
END_VAR
VAR_OUTPUT
	bOK								: BOOL;	// Brak bledow i ostrzezen
	bWarning						: BOOL;	// Ostrzezenie - nie wystepuja w tym podprogramie - wystepuja dla zachowania spojnosci
	bError							: BOOL;	// Zbiorcza flaga bledow
END_VAR
VAR
	bCheckBounds					: BOOL;	// Flaga przekroczen zakresu indexow, np. tablic
	bCheckDivDInt					: BOOL;	// Flaga prob dzielenia Dint przez 0
	bCheckDivLInt					: BOOL; // Flaga prob dzielenia LInt przez 0
	bCheckDivLReal					: BOOL; // Flaga prob dzielenia LREAL przez 0
	bCheckDivReal					: BOOL; // Flaga prob dzielenia REAL przez 0
	bCheckRangeSigned				: BOOL;	// Flaga przekroczen liczby znakowej
	bCheckRangeUnsigned				: BOOL; // Flaga przekroczen liczby bezznakowej
	
	dCheckBoundsOld					: DINT;	// Licznik przekroczen zakresu indexow, np. tablic
	dCheckDivDIntOld				: DINT;	// Licznik prob dzielenia Dint przez 0
	dCheckDivLIntOld				: DINT; // Licznik prob dzielenia LInt przez 0
	dCheckDivLRealOld				: DINT; // Licznik prob dzielenia LREAL przez 0
	dCheckDivRealOld				: DINT; // Licznik prob dzielenia REAL przez 0
	dCheckRangeSignedOld			: DINT;	// Licznik przekroczen  liczby znakowej
	dCheckRangeUnsignedOld			: DINT; // Licznik przekroczen  liczby bezznakowej
END_VAR

IF bReset THEN
	bCheckBounds 					:= FALSE;
	bCheckDivDInt					:= FALSE;
	bCheckDivLInt					:= FALSE;
	bCheckDivLReal					:= FALSE;
	bCheckDivReal					:= FALSE;
	bCheckRangeSigned				:= FALSE;
	bCheckRangeUnsigned				:= FALSE;
ELSE
	bCheckBounds 					S= dCheckBoundsOld <> GVL_Checks.dCheckBounds;
	bCheckDivDInt					S= dCheckDivDIntOld <> GVL_Checks.dCheckDivDInt;
	bCheckDivLInt					S= dCheckDivLIntOld <> GVL_Checks.dCheckDivLInt;
	bCheckDivLReal					S= dCheckDivLRealOld <> GVL_Checks.dCheckDivLReal;
	bCheckDivReal					S= dCheckDivRealOld <> GVL_Checks.dCheckDivReal;
	bCheckRangeSigned				S= dCheckRangeSignedOld <> GVL_Checks.dCheckRangeSigned;
	bCheckRangeUnsigned				S= dCheckRangeUnsignedOld <> GVL_Checks.dCheckRangeUnsigned;	
END_IF

dCheckBoundsOld 					:= GVL_Checks.dCheckBounds;
dCheckDivDIntOld 					:= GVL_Checks.dCheckDivDInt;
dCheckDivLIntOld 					:= GVL_Checks.dCheckDivLInt;
dCheckDivLRealOld 					:= GVL_Checks.dCheckDivLReal;
dCheckDivRealOld 					:= GVL_Checks.dCheckDivReal;
dCheckRangeSignedOld 				:= GVL_Checks.dCheckRangeSigned;
dCheckRangeUnsignedOld 				:= GVL_Checks.dCheckRangeUnsigned;

bError 								:= bCheckBounds OR bCheckDivDInt OR bCheckDivLInt OR bCheckDivLReal OR bCheckDivReal OR bCheckRangeSigned OR bCheckRangeUnsigned;
bOK 								:= NOT bError AND NOT bWarning;

END_PROGRAM

// ---- POUs/Libs/Alarms/VisuEvents/LDT_TO_STRING.TcPOU
FUNCTION LDT_TO_STRING : STRING(24)
VAR_INPUT
	uliTime	:	ULINT; 	//Time [ms]
END_VAR
VAR
	dtTime			:	DATE_AND_TIME;
	uliMillisecond	:	ULINT;
	sTime			:	STRING(24);
END_VAR

IF uliTime = 0 THEN
	LDT_TO_STRING := '-';
	RETURN;
END_IF
dtTime := ULINT_TO_DT(uliTime/1000);
uliMillisecond := uliTime - DT_TO_ULINT(dtTime);
sTime := DT_TO_STRING(dtTime);
sTime := DELETE(sTime,3,1);
sTime := CONCAT(sTime,'.');
if uliMillisecond = 0 then
	sTime := CONCAT(sTime,'000');
ELSIF uliMillisecond < 100 THEN
	sTime := CONCAT(sTime,'0');
	sTime := CONCAT(sTime,ULINT_TO_STRING(uliMillisecond));
ELSE
	sTime := CONCAT(sTime,ULINT_TO_STRING(uliMillisecond));	
END_IF
LDT_TO_STRING := sTime;

END_FUNCTION

// ---- POUs/Libs/Axis/FB_AxisServo.TcPOU
(* 
:Description: This function block is used represent basic axis controled by standard PLCopen motion function blocks.
*)
FUNCTION_BLOCK FB_AxisServo EXTENDS FB_UniversalAxis
VAR
	(* MC_Home *)
	eHomingMode		: MC_HomingMode;		(*  *)
	stHomingOptions	: ST_HomingOptions;		(*  *)
	fbMcHome		: MC_Home;				(*  *)
	
	(* Home switch cam *)
	piHomeSwitch	: FB_DigitalInput;		(*  *)
END_VAR
(*
Version history:

+-------------+------------+----------------+----------+------------------------------------------+
|Date         | Version    | created under  | Author   | Remark                                   |
+=============+============+================+==========+==========================================+
|2021-11      | 1.0.0.0    | V3.1.4024.22   | ADBO     | Function block created                   |
+-------------+------------+----------------+----------+------------------------------------------+

*)

(* Run home switch FB *)
piHomeSwitch();

(* Run parent implementation *)
SUPER^();

PROPERTY HomingMode : MC_HomingMode
GET
HomingMode := eHomingMode;
END_GET
SET
eHomingMode := HomingMode;
END_SET
END_PROPERTY

PROPERTY HomingOptions : ST_HomingOptions
GET
HomingOptions := stHomingOptions;
END_GET
SET
stHomingOptions := HomingOptions;
END_SET
END_PROPERTY

METHOD MR_FirstCycle
VAR_INPUT
	sName 				: STRING; 	(* Axis object name *)
	sMeasurementUnits	: STRING;	(* Measurement units used by axis *)
	bModulo				: BOOL;		(* Axis is periodic *)
END_VAR
SUPER^.MR_FirstCycle(sName:=sName, sMeasurementUnits := sMeasurementUnits, bModulo := bModulo);
piHomeSwitch.MR_FirstCycle(CONCAT(THIS^.sName,', home switch'), sModuleType := piHomeSwitch.ModuleType, sPortID := piHomeSwitch.PortID);
END_METHOD

(* 
Copyrights	: Sonion Industrialization - Control Systems Desing Department
Author		: Adrian Bogdzia - based on MEMS universal libraries
Date		: 11/2021
Description : This function block is used represent basic axis
*)
METHOD PROTECTED MS_Aborting
VAR_INPUT
END_VAR
fbMcHome(Axis := stAxisRef, Execute := FALSE);

SUPER^.MS_Aborting();
END_METHOD

(* 
Copyrights	: Sonion Industrialization - Control Systems Desing Department
Author		: Adrian Bogdzia - based on MEMS universal libraries
Date		: 11/2021
Description : This function block is used represent basic axis
*)
METHOD PROTECTED MS_Halt
VAR_INPUT
END_VAR
(* Reset MC_Home *)
fbMcHome(Axis := stAxisRef, Execute := FALSE);

(* Run parent halt state *)
SUPER^.MS_Halt();
END_METHOD

(* 
Copyrights	: Sonion Industrialization - Control Systems Desing Department
Author		: Adrian Bogdzia - based on MEMS universal libraries
Date		: 11/2021
Description : This function block is used represent basic axis
*)
METHOD PROTECTED MS_Home
VAR_INPUT
END_VAR
fbMcHome(	Axis 			:= stAxisRef,
			Execute 		:= TRUE,
			Position 		:= lrHomePosition,
			HomingMode		:= eHomingMode,
			BufferMode		:= eBufferMode,
			Options			:= stHomingOptions,
			bCalibrationCam := piHomeSwitch.In);
	
IF fbMcHome.Error THEN
	bError := TRUE;
	iErrorID := fbMcHome.ErrorID;
	fbMcHome( Axis := stAxisRef, Execute := FALSE);
	fbAlarmHome.ipArguments.Clear().AddUDInt(iErrorID);	
	fbAlarmHome.Raise(0);
	
ELSIF fbMcHome.Done THEN
	eAxisState := AXIS_HOME_DONE;
		
END_IF
END_METHOD

(* 
Copyrights	: Sonion Industrialization - Control Systems Desing Department
Author		: Adrian Bogdzia - based on MEMS universal libraries
Date		: 11/2021
Description : This function block is used represent basic axis
*)
METHOD PROTECTED MS_HomeDone
VAR_INPUT
END_VAR
fbMcHome(Axis := stAxisRef, Execute := FALSE);

IF NOT bHome AND NOT fbMcHome.Busy THEN
	eAxisState := AXIS_IDLE;
	
END_IF
END_METHOD

(* 
Copyrights	: Sonion Industrialization - Control Systems Desing Department
Author		: Adrian Bogdzia - based on MEMS universal libraries
Date		: 11/2021
Description : This function block is used represent basic axis
*)
METHOD PROTECTED MS_Reset
VAR_INPUT
END_VAR
(* Reset MC_Home*)
fbMcHome( Axis := stAxisRef, Execute := FALSE);

(* Run parent reset procedure*)
IF NOT fbMcHome.Busy THEN
	SUPER^.MS_Reset();
	
END_IF
END_METHOD

(* 
Copyrights	: Precision System Engineering - Control Systems Desing Department
Author		: Adrian Bogdzia - based on MEMS universal libraries
Date		: 11/2021
Description : This function block is used represent basic axis
*)
METHOD PROTECTED MS_Stop
VAR_INPUT
END_VAR
(* Reset MC_Home *)
fbMcHome(Axis := stAxisRef, Execute := FALSE);

(* Run parent stop state *)
SUPER^.MS_Stop();
END_METHOD

PROPERTY ref_HomeSwitch : REFERENCE TO FB_DigitalInput
GET
ref_HomeSwitch REF= piHomeSwitch;
END_GET
END_PROPERTY

END_FUNCTION_BLOCK

// ---- POUs/Libs/Axis/FB_UniversalAxis.TcPOU
(* 
:Description: This function block is base for all other axis devices. It's abstract so it can't be used to create instances.
*)
FUNCTION_BLOCK ABSTRACT FB_UniversalAxis IMPLEMENTS I_UniversalAxis
VAR
	(* Generic *)
	bFirstCycle				: BOOL := TRUE;					(* First cycle bit *)
	sName 					: STRING;						(* Axis name for other utilities *)
	sUnit 					: STRING;						(* Measurement units *)
	bModulo					: BOOL;							(* Axis is periodic *)
	
	(* Hardware link *)
	stAxisRef				: AXIS_REF;						(* Axis reference object *)
	
	(* Internal commands *)
	bInit					: BOOL;							(* Power on axis and prepare to work *)
	bAbort					: BOOL;							(* Power off axis and reset status flags *)
	bHome					: BOOL;							(* Home to reference point *)
	bMoveVelocity			: BOOL;							(* Start motion with constant velocity *)
	bMoveAbsolute			: BOOL;							(* Move to absolute position *)
	bMoveAdditive			: BOOL;							(* Move by distance *)
	bMoveRelative			: BOOL;							(* Move by distance *)
	bJog					: BOOL;							(* Start manual jog movement *)
	bStop					: BOOL;							(* High priority stop command *)
	bHalt					: BOOL;							(* Halt current motion, next motion command will abort this command *)
	bReset					: BOOL;							(* Reset axis and return to READY state *)
	bUnlock					: BOOL;							(* Unlock axis after stop command *)
	//bCouple				: BOOL;							(* Couple appended slave axis *)
	//bDecouple				: BOOL;							(* Decouple appended slave axis *)
	
	(* Internal status - flags *)
	bActive					: BOOL;
	bBusy					: BOOL;							(* Function block currently executes one of the requests *)
	bError					: BOOL;							(* Error status flag *)
	iErrorID				: UDINT;						(* Error ID *)
	iAxisErrorID			: UDINT;						(* Axis error ID *)
	lrActualPosition		: LREAL;						(* Actual axis position in selected units *)
	lrActualVelocity		: LREAL;						(* Actual axis velocity in selected units *)
	bPowerOn 				: BOOL;							(* Power On status bit *)
	bIsHomed				: BOOL;							(* Axis has been homed even once *)
	bInVelocity				: BOOL;							(* Axis is moving in target velocity *)
	bInPostion				: BOOL;							(* Axis reached target position *)
	bMoveActive				: BOOL;							(* Axis is moving to target position *)
	bJogDone				: BOOL;							(* Axis manual movement by jog done *)
	bStopped				: BOOL;							(* Axis movement has been stopped *)
	bHalted					: BOOL;							(* Axis movement has been halted *)
	bLocked					: BOOL;							(* Axis locked after stop commad *)
	eStatePlcOpen			: E_AxisStatePlcOpen;			(* Current PLCOpen state of axis *)
	bHaltLog 				: BOOL;							(* Halt request flag for machine logger *)
	bStopLog 				: BOOL;							(* Stop request flag for machine logger *)
	
	(* Internal status - state machines *)
	eAxisState 				: E_AxisState;					(* Main axis state machine *)
	eAxisStateBeforeReset 	: E_AxisState;					(* State before reset command *)
	eAxisStateInit 			: E_AxisStateInit;				(* Init axis state machine *)
	
	(* General parameters *)
	lrOverride				: LREAL;						(* Axis velocity override in percents [%] *)
	lrVelocity 				: LREAL;						(* Axis velocity in measurement units per second *)
	lrAcceleration			: LREAL;						(* Axis acceleration in measurement units per sercond^2 *)
	lrDeceleration 			: LREAL;						(* Axis deceleration in measurement units per sercond^2 *)
	lrJerk					: LREAL;						(* Axis jerk in measurement unit per sercond^3 *)
	lrAbsolutePosition		: LREAL;						(* Target position for MC_MoveAbsolute function *)
	lrRelativeDistance		: LREAL;						(* Relative distance to move for MC_MoveRelative/Additive fuctions *)
	lrHomePosition			: LREAL;						(* This parameters is used to set axis position while performing homing procedure *)
	
	(* Jog function parameters *)	
	bJogActive				: BOOL;
	lrJogPosition			: LREAL;						(* Relative position to move for jog feature *)
	lrJogVelocity			: LREAL;						(* Jog movement velocity *)
	lrJogAcceleration		: LREAL;						(* Jog movement acceleration *)
	lrJogDeceleration		: LREAL;						(* Jog movement deceleration *)
	lrJogJerk				: LREAL;						(* Jog movement jerk *)
	eJogMode				: E_JogMode;					(* Jog momement mode *)
	eJogDirection			: E_AxisJogDirection;			(* Direction of jog movement *)
	
	(* Stop function parameters *)
	lrStopDeceleration		: LREAL;						(* Stop deceleration *)
	lrStopJerk 				: LREAL;						(* Stop jerk *)
	
	(* Other parameters *)
	stOptions				: ST_MoveOptions;				(* Additional movement options *)
	eDirection				: Tc2_MC2.MC_Direction;			(* Axis movement direction for MC_MoveVelocity *)
	eBufferMode 			: MC_BufferMode := MC_Aborting;	(* Axis buffering mode *)
	
	(* Function blocks - readers *)
	fbReadActualPostion		: MC_ReadActualPosition;		(* FB to read actual position *)
	fbReadActualVelocity	: MC_ReadActualVelocity;		(* FB to read actual velocity *)
	fbReadAxisError			: MC_ReadAxisError;				(* FB to read axis error *)
	fbReadAxisStatus	 	: MC_ReadStatus;				(* FB to read axis status *)
	
	(* Function blocks - administrative *)
	fbMcPower				: MC_Power;						(* FB to control axis power supply and override parameter *)
	fbMcReset				: MC_Reset;						(* FB to reset axis errors *)
	
	(* Function blocks - motion *)
	fbMcMoveVelocity		: MC_MoveVelocity;				(* FB to move axis with constant velocity *)
	fbMcMoveAbsolute		: MC_MoveAbsolute;				(* FB to move axis to absolute postion *)
	fbMcMoveAdditive		: MC_MoveAdditive;				(* FB to move axis by relative distance *)
	fbMcMoveRelative		: MC_MoveRelative;				(* FB to move axis by relative distance *)
	fbMcJog 				: MC_Jog;						(* FB to start axis jog movement *)
	fbMcStop				: MC_Stop;						(* FB to stop axis *)
	fbMcHalt				: MC_Halt;						(* FB to halt axis movement *)
	
	(* Function blocks - linear coupling *)
	fbMcGearIn				: MC_GearIn;					(* FB to couple axis *)		
	fbMcGearOut				: MC_GearOut;					(* FB to decouple axis *)
	
	(* Tc3 EventLogger - messages *)
	fbAlarmHalt 			: FB_TcAlarm;				(*  *)
	fbAlarmInitReset		: FB_TcAlarm;				(*  *)
	fbAlarmInitPowerOn		: FB_TcAlarm;				(*  *)
	fbAlarmMoveAbsolute		: FB_TcAlarm;				(*  *)
	fbAlarmMoveAdditive		: FB_TcAlarm;				(*  *)
	fbAlarmMoveJog			: FB_TcAlarm;				(*  *)	
	fbAlarmMoveRelative		: FB_TcAlarm;				(*  *)	
	fbAlarmMoveVelocity		: FB_TcAlarm;				(*  *)	
	fbAlarmStop				: FB_TcAlarm;				(*  *)
	fbAlarmHome				: FB_TcAlarm;				(*  *)	
	
	fbAlarmHaltCA			: FB_TcAlarm;				(*  *)	
	fbAlarmMoveAbsoluteCA	: FB_TcAlarm;				(*  *)
	fbAlarmMoveRelativeCA	: FB_TcAlarm;				(*  *)
	
	fbAlarmCoupling			: FB_TcAlarm;				(*  *)
	fbAlarmDecoupling		: FB_TcAlarm;				(*  *)		

	bResetConfirmation 		: BOOL;						(*  *)	
	
	rtError					: R_TRIG; 					(* Rising edge trigger for function block error *)

END_VAR


(* Run first cycle procedure *)
IF bFirstCycle THEN
	bFirstCycle := FALSE;
		
	fbAlarmHalt.CreateEx( 	stEventEntry := TC_EVENTS.ShellAxisEventClass.Halt, 
							bWithConfirmation := 1,
							ipSourceInfo := 0);
									
	fbAlarmInitReset.CreateEx( 	stEventEntry := TC_EVENTS.ShellAxisEventClass.InitReset, 
								bWithConfirmation := 1,
								ipSourceInfo := 0);
		
	fbAlarmInitPowerOn.CreateEx( 	stEventEntry := TC_EVENTS.ShellAxisEventClass.InitPowerOn, 
									bWithConfirmation := 1,
									ipSourceInfo := 0);
									
	fbAlarmMoveAbsolute.CreateEx( 	stEventEntry := TC_EVENTS.ShellAxisEventClass.MoveAbsolute, 
									bWithConfirmation := 1,
									ipSourceInfo := 0);
		
	fbAlarmMoveAdditive.CreateEx(	stEventEntry := TC_EVENTS.ShellAxisEventClass.MoveAdditive, 
									bWithConfirmation := 1,
									ipSourceInfo := 0);
									
	fbAlarmMoveJog.CreateEx( 	stEventEntry := TC_EVENTS.ShellAxisEventClass.MoveJog, 
								bWithConfirmation := 1,
								ipSourceInfo := 0);
		
	fbAlarmMoveRelative.CreateEx( stEventEntry := TC_EVENTS.ShellAxisEventClass.MoveRelative, 
									bWithConfirmation := 1,
									ipSourceInfo := 0);
									
	fbAlarmMoveVelocity.CreateEx(	stEventEntry := TC_EVENTS.ShellAxisEventClass.MoveVelocity, 
									bWithConfirmation := 1,
									ipSourceInfo := 0);
		
	fbAlarmStop.CreateEx( 	stEventEntry := TC_EVENTS.ShellAxisEventClass.Stop, 
							bWithConfirmation := 1,
							ipSourceInfo := 0);
									
	fbAlarmHome.CreateEx( 	stEventEntry := TC_EVENTS.ShellAxisEventClass.Home, 
							bWithConfirmation := 1,
							ipSourceInfo := 0);									

	fbAlarmHaltCA.CreateEx( stEventEntry := TC_EVENTS.ShellAxisEventClass.HaltCA, 
							bWithConfirmation := 1,
							ipSourceInfo := 0);
		
	fbAlarmMoveAbsoluteCA.CreateEx( stEventEntry := TC_EVENTS.ShellAxisEventClass.MoveAbsoluteCA, 
									bWithConfirmation := 1,
									ipSourceInfo := 0);
									
	fbAlarmMoveRelativeCA.CreateEx( stEventEntry := TC_EVENTS.ShellAxisEventClass.MoveRelativeCA, 
									bWithConfirmation := 1,
									ipSourceInfo := 0);
		
	fbAlarmCoupling.CreateEx( stEventEntry := TC_EVENTS.ShellAxisEventClass.Coupling, 
									bWithConfirmation := 1,
									ipSourceInfo := 0);
									
	fbAlarmDecoupling.CreateEx( stEventEntry := TC_EVENTS.ShellAxisEventClass.Decoupling, 
									bWithConfirmation := 1,
									ipSourceInfo := 0);									
									
END_IF

(* Read AXIS_REF status *)
stAxisRef.ReadStatus();

(* Read axis PLCOpen state *)
fbReadAxisStatus( Axis := stAxisRef, Enable := TRUE);
					
IF fbReadAxisStatus.Valid THEN
	IF fbReadAxisStatus.Disabled THEN
		eStatePlcOpen := AXIS_PLCOPEN_DISABLED;
		
	ELSIF fbReadAxisStatus.StandStill THEN
		eStatePlcOpen := AXIS_PLCOPEN_STANDSTILL;
		
	ELSIF fbReadAxisStatus.Homing THEN
		eStatePlcOpen := AXIS_PLCOPEN_HOMING;
		
	ELSIF fbReadAxisStatus.DiscreteMotion THEN
		eStatePlcOpen := AXIS_PLCOPEN_DISCRETE_MOTION;
		
	ELSIF fbReadAxisStatus.ContinuousMotion THEN
		eStatePlcOpen := AXIS_PLCOPEN_CONTINUOUS_MOTION;
		
	ELSIF fbReadAxisStatus.SynchronizedMotion THEN
		eStatePlcOpen := AXIS_PLCOPEN_SYNCHRONIZED_MOTION;
		
	ELSIF fbReadAxisStatus.ErrorStop THEN
		eStatePlcOpen := AXIS_PLCOPEN_ERRORSTOP;
		
	END_IF
END_IF

(* Update status flags *)
bActive := (eAxisState >= AXIS_READY_INITIALIZED);
bBusy := eAxisState <> AXIS_UNINITIALIZED AND eAxisState <> AXIS_IDLE;
bPowerOn := NOT stAxisRef.Status.Disabled;

(* Read axis errors *)
fbReadAxisError(	Axis := stAxisRef,
					Enable := TRUE,
					AxisErrorID => iAxisErrorID);

(* Read actual axis postion *)
IF bModulo THEN
	lrActualPosition := stAxisRef.NcToPlc.ModuloActPos;
ELSE
	fbReadActualPostion(	Axis := stAxisRef,
							Enable := TRUE,
							Position => lrActualPosition);
END_IF


(* Read actual axis velocity *)
fbReadActualVelocity( 	Axis := stAxisRef,
						Enable := TRUE,
						ActualVelocity => lrActualVelocity);		

(* Report errors that occur *)
rtError(CLK:=bError);

IF rtError.Q THEN 
	fbMachineLogger.MR_AddLogs(FUN_MergeStrings5(sName, ' : Error occured (error ID: ', UDINT_TO_STRING(iErrorID), ')', ''));

END_IF
						
(* Execute main state machine *)
StateMachine();

PROPERTY Acceleration : LREAL
GET
Acceleration := lrAcceleration;
END_GET
SET
lrAcceleration := Acceleration;
END_SET
END_PROPERTY

PROPERTY Active : REFERENCE TO BOOL
GET
Active REF= bActive;
END_GET
END_PROPERTY

PROPERTY ActualPosition : REFERENCE TO LREAL
GET
ActualPosition REF= lrActualPosition;
END_GET
END_PROPERTY

